  PROC DrawPart12()
    MoveL Offs(pOrigin,319.92,43.79,0.00),v40,z0,tPen\WObj:=wPaper;
    MoveL Offs(pOrigin,319.60,42.83,0.00),v40,z0,tPen\WObj:=wPaper;
    MoveL Offs(pOrigin,310.98,31.34,0.00),v40,z0,tPen\WObj:=wPaper;
    MoveL Offs(pOrigin,310.98,30.86,0.00),v40,z0,tPen\WObj:=wPaper;
    MoveL Offs(pOrigin,311.77,30.38,0.00),v40,z0,tPen\WObj:=wPaper;
    MoveL Offs(pOrigin,318.48,30.38,0.00),v40,z0,tPen\WObj:=wPaper;
    MoveL Offs(pOrigin,319.44,30.06,0.00),v40,z0,tPen\WObj:=wPaper;
    MoveL Offs(pOrigin,319.92,29.42,0.00),v40,z0,tPen\WObj:=wPaper;
    MoveL Offs(pOrigin,319.92,27.51,0.00),v40,z0,tPen\WObj:=wPaper;
    MoveL Offs(pOrigin,319.44,26.87,0.00),v40,z0,tPen\WObj:=wPaper;
    MoveL Offs(pOrigin,318.48,26.55,0.00),v40,z0,tPen\WObj:=wPaper;
    MoveL Offs(pOrigin,306.51,26.55,0.00),v40,z0,tPen\WObj:=wPaper;
    MoveL Offs(pOrigin,304.75,27.19,0.00),v40,z0,tPen\WObj:=wPaper;
    MoveL Offs(pOrigin,304.75,29.90,0.00),v40,z0,tPen\WObj:=wPaper;
    MoveL Offs(pOrigin,313.85,41.87,0.00),v40,z0,tPen\WObj:=wPaper;
    MoveL Offs(pOrigin,313.69,42.67,0.00),v40,z0,tPen\WObj:=wPaper;
    MoveL Offs(pOrigin,310.34,42.83,0.00),v40,z0,tPen\WObj:=wPaper;
    MoveL Offs(pOrigin,308.90,43.31,0.00),v40,z0,tPen\WObj:=wPaper;
    MoveL Offs(pOrigin,305.71,43.47,0.00),v40,z0,tPen\WObj:=wPaper;
    MoveL Offs(pOrigin,305.07,44.75,0.00),v40,fine,tPen\WObj:=wPaper;
    MoveL Offs(pOrigin,305.07,44.75,6.00),v60,z5,tPen\WObj:=wPaper;
    MoveL Offs(pOrigin,312.25,39.96,6.00),vTravel,z5,tPen\WObj:=wPaper;
    MoveL Offs(pOrigin,312.25,39.96,0.00),v60,z0,tPen\WObj:=wPaper;
    MoveL Offs(pOrigin,312.73,39.96,0.00),v40,z0,tPen\WObj:=wPaper;
    MoveL Offs(pOrigin,313.69,40.92,0.00),v40,z0,tPen\WObj:=wPaper;
    MoveL Offs(pOrigin,312.25,39.48,0.00),v40,z0,tPen\WObj:=wPaper;
    MoveL Offs(pOrigin,312.25,39.96,0.00),v40,z0,tPen\WObj:=wPaper;
    MoveL Offs(pOrigin,312.73,39.96,0.00),v40,z0,tPen\WObj:=wPaper;
    MoveL Offs(pOrigin,313.69,40.92,0.00),v40,z0,tPen\WObj:=wPaper;
    MoveL Offs(pOrigin,312.25,39.48,0.00),v40,z0,tPen\WObj:=wPaper;
    MoveL Offs(pOrigin,312.25,39.96,0.00),v40,fine,tPen\WObj:=wPaper;
    MoveL Offs(pOrigin,312.25,39.96,6.00),v60,z5,tPen\WObj:=wPaper;
    MoveL Offs(pOrigin,311.77,38.52,6.00),vTravel,z5,tPen\WObj:=wPaper;
    MoveL Offs(pOrigin,311.77,38.52,0.00),v60,z0,tPen\WObj:=wPaper;
    MoveL Offs(pOrigin,311.30,38.04,0.00),v40,z0,tPen\WObj:=wPaper;
    MoveL Offs(pOrigin,311.30,38.52,0.00),v40,z0,tPen\WObj:=wPaper;
    MoveL Offs(pOrigin,311.77,38.52,0.00),v40,z0,tPen\WObj:=wPaper;
    MoveL Offs(pOrigin,311.30,38.04,0.00),v40,z0,tPen\WObj:=wPaper;
    MoveL Offs(pOrigin,311.30,38.52,0.00),v40,z0,tPen\WObj:=wPaper;
    MoveL Offs(pOrigin,311.77,38.52,0.00),v40,fine,tPen\WObj:=wPaper;
    MoveL Offs(pOrigin,311.77,38.52,6.00),v60,z5,tPen\WObj:=wPaper;
    MoveL Offs(pOrigin,310.82,37.08,6.00),vTravel,z5,tPen\WObj:=wPaper;
    MoveL Offs(pOrigin,310.82,37.08,0.00),v60,z0,tPen\WObj:=wPaper;
    MoveL Offs(pOrigin,310.34,36.61,0.00),v40,z0,tPen\WObj:=wPaper;
    MoveL Offs(pOrigin,310.34,37.08,0.00),v40,z0,tPen\WObj:=wPaper;
    MoveL Offs(pOrigin,310.82,37.08,0.00),v40,z0,tPen\WObj:=wPaper;
    MoveL Offs(pOrigin,310.34,36.61,0.00),v40,z0,tPen\WObj:=wPaper;
    MoveL Offs(pOrigin,310.34,37.08,0.00),v40,z0,tPen\WObj:=wPaper;
    MoveL Offs(pOrigin,310.82,37.08,0.00),v40,fine,tPen\WObj:=wPaper;
    MoveL Offs(pOrigin,310.82,37.08,6.00),v60,z5,tPen\WObj:=wPaper;
    MoveL Offs(pOrigin,309.86,35.65,6.00),vTravel,z5,tPen\WObj:=wPaper;
    MoveL Offs(pOrigin,309.86,35.65,0.00),v60,z0,tPen\WObj:=wPaper;
    MoveL Offs(pOrigin,309.38,35.17,0.00),v40,z0,tPen\WObj:=wPaper;
    MoveL Offs(pOrigin,309.38,35.65,0.00),v40,z0,tPen\WObj:=wPaper;
    MoveL Offs(pOrigin,309.86,35.65,0.00),v40,z0,tPen\WObj:=wPaper;
    MoveL Offs(pOrigin,309.38,35.17,0.00),v40,z0,tPen\WObj:=wPaper;
    MoveL Offs(pOrigin,309.38,35.65,0.00),v40,z0,tPen\WObj:=wPaper;
    MoveL Offs(pOrigin,309.86,35.65,0.00),v40,fine,tPen\WObj:=wPaper;
    MoveL Offs(pOrigin,309.86,35.65,6.00),v60,z5,tPen\WObj:=wPaper;
    MoveL Offs(pOrigin,312.25,33.73,6.00),vTravel,z5,tPen\WObj:=wPaper;
    MoveL Offs(pOrigin,312.25,33.73,0.00),v60,z0,tPen\WObj:=wPaper;
    MoveL Offs(pOrigin,313.21,34.69,0.00),v40,z0,tPen\WObj:=wPaper;
    MoveL Offs(pOrigin,312.25,33.73,0.00),v40,z0,tPen\WObj:=wPaper;
    MoveL Offs(pOrigin,311.77,33.25,0.00),v40,z0,tPen\WObj:=wPaper;
    MoveL Offs(pOrigin,311.30,32.30,0.00),v40,z0,tPen\WObj:=wPaper;
    MoveL Offs(pOrigin,311.77,32.77,0.00),v40,z0,tPen\WObj:=wPaper;
    MoveL Offs(pOrigin,311.77,33.25,0.00),v40,z0,tPen\WObj:=wPaper;
    MoveL Offs(pOrigin,311.30,32.30,0.00),v40,z0,tPen\WObj:=wPaper;
    MoveL Offs(pOrigin,311.77,32.77,0.00),v40,z0,tPen\WObj:=wPaper;
    MoveL Offs(pOrigin,311.77,33.25,0.00),v40,fine,tPen\WObj:=wPaper;
    MoveL Offs(pOrigin,311.77,33.25,6.00),v60,z5,tPen\WObj:=wPaper;
    MoveL Offs(pOrigin,314.17,36.13,6.00),vTravel,z5,tPen\WObj:=wPaper;
    MoveL Offs(pOrigin,314.17,36.13,0.00),v60,z0,tPen\WObj:=wPaper;
    MoveL Offs(pOrigin,314.65,36.61,0.00),v40,z0,tPen\WObj:=wPaper;
    MoveL Offs(pOrigin,314.65,37.08,0.00),v40,z0,tPen\WObj:=wPaper;
    MoveL Offs(pOrigin,316.08,38.52,0.00),v40,z0,tPen\WObj:=wPaper;
    MoveL Offs(pOrigin,314.17,36.13,0.00),v40,z0,tPen\WObj:=wPaper;
    MoveL Offs(pOrigin,314.65,36.61,0.00),v40,z0,tPen\WObj:=wPaper;
    MoveL Offs(pOrigin,314.65,37.08,0.00),v40,z0,tPen\WObj:=wPaper;
    MoveL Offs(pOrigin,316.08,38.52,0.00),v40,z0,tPen\WObj:=wPaper;
    MoveL Offs(pOrigin,314.17,36.13,0.00),v40,fine,tPen\WObj:=wPaper;
    MoveL Offs(pOrigin,314.17,36.13,6.00),v60,z5,tPen\WObj:=wPaper;
    MoveL Offs(pOrigin,317.52,40.92,6.00),vTravel,z5,tPen\WObj:=wPaper;
    MoveL Offs(pOrigin,317.52,40.92,0.00),v60,z0,tPen\WObj:=wPaper;
    MoveL Offs(pOrigin,318.96,42.35,0.00),v40,z0,tPen\WObj:=wPaper;
    MoveL Offs(pOrigin,317.52,40.92,0.00),v40,fine,tPen\WObj:=wPaper;
    MoveL Offs(pOrigin,317.52,40.92,6.00),v60,z5,tPen\WObj:=wPaper;
    MoveL Offs(pOrigin,307.94,33.25,6.00),vTravel,z5,tPen\WObj:=wPaper;
    MoveL Offs(pOrigin,307.94,33.25,0.00),v60,z0,tPen\WObj:=wPaper;
    MoveL Offs(pOrigin,306.99,32.30,0.00),v40,z0,tPen\WObj:=wPaper;
    MoveL Offs(pOrigin,306.99,32.77,0.00),v40,z0,tPen\WObj:=wPaper;
    MoveL Offs(pOrigin,307.46,32.77,0.00),v40,z0,tPen\WObj:=wPaper;
    MoveL Offs(pOrigin,307.94,33.25,0.00),v40,z0,tPen\WObj:=wPaper;
    MoveL Offs(pOrigin,306.99,32.30,0.00),v40,z0,tPen\WObj:=wPaper;
    MoveL Offs(pOrigin,306.99,32.77,0.00),v40,z0,tPen\WObj:=wPaper;
    MoveL Offs(pOrigin,307.46,32.77,0.00),v40,z0,tPen\WObj:=wPaper;
    MoveL Offs(pOrigin,307.94,33.25,0.00),v40,fine,tPen\WObj:=wPaper;
    MoveL Offs(pOrigin,307.94,33.25,6.00),v60,z5,tPen\WObj:=wPaper;
    MoveL Offs(pOrigin,306.51,31.34,6.00),vTravel,z5,tPen\WObj:=wPaper;
    MoveL Offs(pOrigin,306.51,31.34,0.00),v60,z0,tPen\WObj:=wPaper;
    MoveL Offs(pOrigin,306.03,30.86,0.00),v40,z0,tPen\WObj:=wPaper;
    MoveL Offs(pOrigin,306.03,31.34,0.00),v40,z0,tPen\WObj:=wPaper;
    MoveL Offs(pOrigin,306.51,31.34,0.00),v40,z0,tPen\WObj:=wPaper;
    MoveL Offs(pOrigin,306.03,30.86,0.00),v40,z0,tPen\WObj:=wPaper;
    MoveL Offs(pOrigin,306.03,31.34,0.00),v40,z0,tPen\WObj:=wPaper;
    MoveL Offs(pOrigin,306.51,31.34,0.00),v40,fine,tPen\WObj:=wPaper;
    MoveL Offs(pOrigin,306.51,31.34,6.00),v60,z5,tPen\WObj:=wPaper;
    MoveL Offs(pOrigin,329.01,28.46,6.00),vTravel,z5,tPen\WObj:=wPaper;
    MoveL Offs(pOrigin,329.01,28.46,0.00),v60,z0,tPen\WObj:=wPaper;
    MoveL Offs(pOrigin,333.48,39.00,0.00),v40,z0,tPen\WObj:=wPaper;
    MoveL Offs(pOrigin,334.12,41.39,0.00),v40,z0,tPen\WObj:=wPaper;
    MoveL Offs(pOrigin,335.88,45.23,0.00),v40,z0,tPen\WObj:=wPaper;
    MoveL Offs(pOrigin,337.15,46.34,0.00),v40,z0,tPen\WObj:=wPaper;
    MoveL Offs(pOrigin,339.55,46.66,0.00),v40,z0,tPen\WObj:=wPaper;
    MoveL Offs(pOrigin,340.83,45.70,0.00),v40,z0,tPen\WObj:=wPaper;
    MoveL Offs(pOrigin,346.41,31.82,0.00),v40,z0,tPen\WObj:=wPaper;
    MoveL Offs(pOrigin,347.69,27.99,0.00),v40,z0,tPen\WObj:=wPaper;
    MoveL Offs(pOrigin,347.21,26.87,0.00),v40,z0,tPen\WObj:=wPaper;
    MoveL Offs(pOrigin,345.77,26.55,0.00),v40,z0,tPen\WObj:=wPaper;
    MoveL Offs(pOrigin,344.34,27.19,0.00),v40,z0,tPen\WObj:=wPaper;
  ENDPROC

  PROC DrawPart13()
    MoveL Offs(pOrigin,343.06,29.90,0.00),v40,z0,tPen\WObj:=wPaper;
    MoveL Offs(pOrigin,342.42,30.38,0.00),v40,z0,tPen\WObj:=wPaper;
    MoveL Offs(pOrigin,340.03,30.38,0.00),v40,z0,tPen\WObj:=wPaper;
    MoveL Offs(pOrigin,338.59,30.86,0.00),v40,z0,tPen\WObj:=wPaper;
    MoveL Offs(pOrigin,335.72,30.86,0.00),v40,z0,tPen\WObj:=wPaper;
    MoveL Offs(pOrigin,333.80,29.90,0.00),v40,z0,tPen\WObj:=wPaper;
    MoveL Offs(pOrigin,332.69,27.51,0.00),v40,z0,tPen\WObj:=wPaper;
    MoveL Offs(pOrigin,331.89,26.87,0.00),v40,z0,tPen\WObj:=wPaper;
    MoveL Offs(pOrigin,330.45,26.55,0.00),v40,z0,tPen\WObj:=wPaper;
    MoveL Offs(pOrigin,329.17,27.19,0.00),v40,z0,tPen\WObj:=wPaper;
    MoveL Offs(pOrigin,329.01,28.46,0.00),v40,fine,tPen\WObj:=wPaper;
    MoveL Offs(pOrigin,329.01,28.46,6.00),v60,z5,tPen\WObj:=wPaper;
    MoveL Offs(pOrigin,331.41,33.73,6.00),vTravel,z5,tPen\WObj:=wPaper;
    MoveL Offs(pOrigin,331.41,33.73,0.00),v60,z0,tPen\WObj:=wPaper;
    MoveL Offs(pOrigin,331.41,34.21,0.00),v40,z0,tPen\WObj:=wPaper;
    MoveL Offs(pOrigin,331.89,34.69,0.00),v40,z0,tPen\WObj:=wPaper;
    MoveL Offs(pOrigin,331.41,33.73,0.00),v40,z0,tPen\WObj:=wPaper;
    MoveL Offs(pOrigin,331.41,34.21,0.00),v40,z0,tPen\WObj:=wPaper;
    MoveL Offs(pOrigin,331.89,34.69,0.00),v40,z0,tPen\WObj:=wPaper;
    MoveL Offs(pOrigin,331.41,33.73,0.00),v40,fine,tPen\WObj:=wPaper;
    MoveL Offs(pOrigin,331.41,33.73,6.00),v60,z5,tPen\WObj:=wPaper;
    MoveL Offs(pOrigin,335.72,34.21,6.00),vTravel,z5,tPen\WObj:=wPaper;
    MoveL Offs(pOrigin,335.72,34.21,0.00),v60,z0,tPen\WObj:=wPaper;
    MoveL Offs(pOrigin,335.72,35.17,0.00),v40,z0,tPen\WObj:=wPaper;
    MoveL Offs(pOrigin,337.79,40.44,0.00),v40,z0,tPen\WObj:=wPaper;
    MoveL Offs(pOrigin,338.59,40.76,0.00),v40,z0,tPen\WObj:=wPaper;
    MoveL Offs(pOrigin,339.55,39.48,0.00),v40,z0,tPen\WObj:=wPaper;
    MoveL Offs(pOrigin,340.51,36.13,0.00),v40,z0,tPen\WObj:=wPaper;
    MoveL Offs(pOrigin,340.51,34.69,0.00),v40,z0,tPen\WObj:=wPaper;
    MoveL Offs(pOrigin,340.03,34.05,0.00),v40,z0,tPen\WObj:=wPaper;
    MoveL Offs(pOrigin,339.07,33.73,0.00),v40,z0,tPen\WObj:=wPaper;
    MoveL Offs(pOrigin,336.20,33.73,0.00),v40,z0,tPen\WObj:=wPaper;
    MoveL Offs(pOrigin,335.72,34.21,0.00),v40,fine,tPen\WObj:=wPaper;
    MoveL Offs(pOrigin,335.72,34.21,6.00),v60,z5,tPen\WObj:=wPaper;
    MoveL Offs(pOrigin,314.65,83.06,6.00),vTravel,z5,tPen\WObj:=wPaper;
    MoveL Offs(pOrigin,314.65,83.06,0.00),v60,z0,tPen\WObj:=wPaper;
    MoveL Offs(pOrigin,314.65,83.54,0.00),v40,z0,tPen\WObj:=wPaper;
    MoveL Offs(pOrigin,315.13,83.54,0.00),v40,z0,tPen\WObj:=wPaper;
    MoveL Offs(pOrigin,314.65,83.06,0.00),v40,z0,tPen\WObj:=wPaper;
    MoveL Offs(pOrigin,314.65,83.54,0.00),v40,z0,tPen\WObj:=wPaper;
    MoveL Offs(pOrigin,315.13,83.54,0.00),v40,z0,tPen\WObj:=wPaper;
    MoveL Offs(pOrigin,314.65,83.06,0.00),v40,fine,tPen\WObj:=wPaper;
    MoveL Offs(pOrigin,314.65,83.06,6.00),v60,z5,tPen\WObj:=wPaper;
    MoveL Offs(pOrigin,319.92,86.89,6.00),vTravel,z5,tPen\WObj:=wPaper;
    MoveL Offs(pOrigin,319.92,86.89,0.00),v60,z0,tPen\WObj:=wPaper;
    MoveL Offs(pOrigin,319.92,87.37,0.00),v40,z0,tPen\WObj:=wPaper;
    MoveL Offs(pOrigin,320.39,87.37,0.00),v40,z0,tPen\WObj:=wPaper;
    MoveL Offs(pOrigin,319.92,86.89,0.00),v40,z0,tPen\WObj:=wPaper;
    MoveL Offs(pOrigin,319.92,87.37,0.00),v40,z0,tPen\WObj:=wPaper;
    MoveL Offs(pOrigin,320.39,87.37,0.00),v40,z0,tPen\WObj:=wPaper;
    MoveL Offs(pOrigin,319.92,86.89,0.00),v40,fine,tPen\WObj:=wPaper;
    MoveL Offs(pOrigin,319.92,86.89,6.00),v60,z5,tPen\WObj:=wPaper;
    MoveL Offs(pOrigin,322.79,88.80,6.00),vTravel,z5,tPen\WObj:=wPaper;
    MoveL Offs(pOrigin,322.79,88.80,0.00),v60,z0,tPen\WObj:=wPaper;
    MoveL Offs(pOrigin,322.79,89.28,0.00),v40,z0,tPen\WObj:=wPaper;
    MoveL Offs(pOrigin,323.27,89.28,0.00),v40,z0,tPen\WObj:=wPaper;
    MoveL Offs(pOrigin,324.23,90.24,0.00),v40,z0,tPen\WObj:=wPaper;
    MoveL Offs(pOrigin,322.79,88.80,0.00),v40,z0,tPen\WObj:=wPaper;
    MoveL Offs(pOrigin,322.79,89.28,0.00),v40,z0,tPen\WObj:=wPaper;
    MoveL Offs(pOrigin,323.27,89.28,0.00),v40,z0,tPen\WObj:=wPaper;
    MoveL Offs(pOrigin,324.23,90.24,0.00),v40,z0,tPen\WObj:=wPaper;
    MoveL Offs(pOrigin,322.79,88.80,0.00),v40,fine,tPen\WObj:=wPaper;
    MoveL Offs(pOrigin,322.79,88.80,6.00),v60,z5,tPen\WObj:=wPaper;
    MoveL Offs(pOrigin,325.66,91.20,6.00),vTravel,z5,tPen\WObj:=wPaper;
    MoveL Offs(pOrigin,325.66,91.20,0.00),v60,z0,tPen\WObj:=wPaper;
    MoveL Offs(pOrigin,325.66,91.68,0.00),v40,z0,tPen\WObj:=wPaper;
    MoveL Offs(pOrigin,326.14,91.68,0.00),v40,z0,tPen\WObj:=wPaper;
    MoveL Offs(pOrigin,326.62,92.15,0.00),v40,z0,tPen\WObj:=wPaper;
    MoveL Offs(pOrigin,325.66,91.20,0.00),v40,z0,tPen\WObj:=wPaper;
    MoveL Offs(pOrigin,325.66,91.68,0.00),v40,z0,tPen\WObj:=wPaper;
    MoveL Offs(pOrigin,326.14,91.68,0.00),v40,z0,tPen\WObj:=wPaper;
    MoveL Offs(pOrigin,326.62,92.15,0.00),v40,z0,tPen\WObj:=wPaper;
    MoveL Offs(pOrigin,325.66,91.20,0.00),v40,fine,tPen\WObj:=wPaper;
    MoveL Offs(pOrigin,325.66,91.20,6.00),v60,z5,tPen\WObj:=wPaper;
    MoveL Offs(pOrigin,329.01,94.07,6.00),vTravel,z5,tPen\WObj:=wPaper;
    MoveL Offs(pOrigin,329.01,94.07,0.00),v60,z0,tPen\WObj:=wPaper;
    MoveL Offs(pOrigin,329.01,94.55,0.00),v40,z0,tPen\WObj:=wPaper;
    MoveL Offs(pOrigin,329.49,94.55,0.00),v40,z0,tPen\WObj:=wPaper;
    MoveL Offs(pOrigin,329.97,95.03,0.00),v40,z0,tPen\WObj:=wPaper;
    MoveL Offs(pOrigin,329.01,94.07,0.00),v40,z0,tPen\WObj:=wPaper;
    MoveL Offs(pOrigin,329.01,94.55,0.00),v40,z0,tPen\WObj:=wPaper;
    MoveL Offs(pOrigin,329.49,94.55,0.00),v40,z0,tPen\WObj:=wPaper;
    MoveL Offs(pOrigin,329.97,95.03,0.00),v40,z0,tPen\WObj:=wPaper;
    MoveL Offs(pOrigin,329.01,94.07,0.00),v40,fine,tPen\WObj:=wPaper;
    MoveL Offs(pOrigin,329.01,94.07,6.00),v60,z5,tPen\WObj:=wPaper;
    MoveL Offs(pOrigin,331.09,95.83,6.00),vTravel,z5,tPen\WObj:=wPaper;
    MoveL Offs(pOrigin,331.09,95.83,0.00),v60,z0,tPen\WObj:=wPaper;
    MoveL Offs(pOrigin,335.24,99.82,0.00),v40,z0,tPen\WObj:=wPaper;
    MoveL Offs(pOrigin,331.09,95.83,0.00),v40,fine,tPen\WObj:=wPaper;
    MoveL Offs(pOrigin,331.09,95.83,6.00),v60,z5,tPen\WObj:=wPaper;
    MoveL Offs(pOrigin,336.68,101.25,6.00),vTravel,z5,tPen\WObj:=wPaper;
    MoveL Offs(pOrigin,336.68,101.25,0.00),v60,z0,tPen\WObj:=wPaper;
    MoveL Offs(pOrigin,336.68,101.73,0.00),v40,z0,tPen\WObj:=wPaper;
    MoveL Offs(pOrigin,337.15,101.73,0.00),v40,z0,tPen\WObj:=wPaper;
    MoveL Offs(pOrigin,340.03,104.61,0.00),v40,z0,tPen\WObj:=wPaper;
    MoveL Offs(pOrigin,336.68,101.25,0.00),v40,z0,tPen\WObj:=wPaper;
    MoveL Offs(pOrigin,336.68,101.73,0.00),v40,z0,tPen\WObj:=wPaper;
    MoveL Offs(pOrigin,337.15,101.73,0.00),v40,z0,tPen\WObj:=wPaper;
    MoveL Offs(pOrigin,340.03,104.61,0.00),v40,z0,tPen\WObj:=wPaper;
    MoveL Offs(pOrigin,336.68,101.25,0.00),v40,fine,tPen\WObj:=wPaper;
    MoveL Offs(pOrigin,336.68,101.25,6.00),v60,z5,tPen\WObj:=wPaper;
    MoveL Offs(pOrigin,340.51,105.08,6.00),vTravel,z5,tPen\WObj:=wPaper;
    MoveL Offs(pOrigin,340.51,105.08,0.00),v60,z0,tPen\WObj:=wPaper;
    MoveL Offs(pOrigin,340.51,105.56,0.00),v40,z0,tPen\WObj:=wPaper;
    MoveL Offs(pOrigin,340.99,105.56,0.00),v40,z0,tPen\WObj:=wPaper;
    MoveL Offs(pOrigin,341.94,106.52,0.00),v40,z0,tPen\WObj:=wPaper;
    MoveL Offs(pOrigin,340.51,105.08,0.00),v40,z0,tPen\WObj:=wPaper;
    MoveL Offs(pOrigin,340.51,105.56,0.00),v40,z0,tPen\WObj:=wPaper;
    MoveL Offs(pOrigin,340.99,105.56,0.00),v40,z0,tPen\WObj:=wPaper;
    MoveL Offs(pOrigin,341.94,106.52,0.00),v40,z0,tPen\WObj:=wPaper;
    MoveL Offs(pOrigin,340.51,105.08,0.00),v40,fine,tPen\WObj:=wPaper;
    MoveL Offs(pOrigin,340.51,105.08,6.00),v60,z5,tPen\WObj:=wPaper;
    MoveL Offs(pOrigin,342.90,107.96,6.00),vTravel,z5,tPen\WObj:=wPaper;
    MoveL Offs(pOrigin,342.90,107.96,0.00),v60,z0,tPen\WObj:=wPaper;
    MoveL Offs(pOrigin,342.90,108.44,0.00),v40,z0,tPen\WObj:=wPaper;
    MoveL Offs(pOrigin,343.38,108.44,0.00),v40,z0,tPen\WObj:=wPaper;
    MoveL Offs(pOrigin,343.86,108.92,0.00),v40,z0,tPen\WObj:=wPaper;
    MoveL Offs(pOrigin,342.90,107.96,0.00),v40,z0,tPen\WObj:=wPaper;
    MoveL Offs(pOrigin,342.90,108.44,0.00),v40,z0,tPen\WObj:=wPaper;
    MoveL Offs(pOrigin,343.38,108.44,0.00),v40,z0,tPen\WObj:=wPaper;
  ENDPROC

  PROC DrawPart14()
    MoveL Offs(pOrigin,343.86,108.92,0.00),v40,z0,tPen\WObj:=wPaper;
    MoveL Offs(pOrigin,342.90,107.96,0.00),v40,fine,tPen\WObj:=wPaper;
    MoveL Offs(pOrigin,342.90,107.96,6.00),v60,z5,tPen\WObj:=wPaper;
    MoveL Offs(pOrigin,345.77,111.31,6.00),vTravel,z5,tPen\WObj:=wPaper;
    MoveL Offs(pOrigin,345.77,111.31,0.00),v60,z0,tPen\WObj:=wPaper;
    MoveL Offs(pOrigin,345.77,111.79,0.00),v40,z0,tPen\WObj:=wPaper;
    MoveL Offs(pOrigin,347.21,113.23,0.00),v40,z0,tPen\WObj:=wPaper;
    MoveL Offs(pOrigin,345.77,111.31,0.00),v40,z0,tPen\WObj:=wPaper;
    MoveL Offs(pOrigin,345.77,111.79,0.00),v40,z0,tPen\WObj:=wPaper;
    MoveL Offs(pOrigin,347.21,113.23,0.00),v40,z0,tPen\WObj:=wPaper;
    MoveL Offs(pOrigin,345.77,111.31,0.00),v40,fine,tPen\WObj:=wPaper;
    MoveL Offs(pOrigin,345.77,111.31,6.00),v60,z5,tPen\WObj:=wPaper;
    MoveL Offs(pOrigin,347.69,113.70,6.00),vTravel,z5,tPen\WObj:=wPaper;
    MoveL Offs(pOrigin,347.69,113.70,0.00),v60,z0,tPen\WObj:=wPaper;
    MoveL Offs(pOrigin,347.69,114.18,0.00),v40,z0,tPen\WObj:=wPaper;
    MoveL Offs(pOrigin,348.65,115.14,0.00),v40,z0,tPen\WObj:=wPaper;
    MoveL Offs(pOrigin,347.69,113.70,0.00),v40,z0,tPen\WObj:=wPaper;
    MoveL Offs(pOrigin,347.69,114.18,0.00),v40,z0,tPen\WObj:=wPaper;
    MoveL Offs(pOrigin,348.65,115.14,0.00),v40,z0,tPen\WObj:=wPaper;
    MoveL Offs(pOrigin,347.69,113.70,0.00),v40,fine,tPen\WObj:=wPaper;
    MoveL Offs(pOrigin,347.69,113.70,6.00),v60,z5,tPen\WObj:=wPaper;
    MoveL Offs(pOrigin,349.13,116.10,6.00),vTravel,z5,tPen\WObj:=wPaper;
    MoveL Offs(pOrigin,349.13,116.10,0.00),v60,z0,tPen\WObj:=wPaper;
    MoveL Offs(pOrigin,349.13,116.58,0.00),v40,z0,tPen\WObj:=wPaper;
    MoveL Offs(pOrigin,349.61,116.58,0.00),v40,z0,tPen\WObj:=wPaper;
    MoveL Offs(pOrigin,350.08,117.06,0.00),v40,z0,tPen\WObj:=wPaper;
    MoveL Offs(pOrigin,349.13,116.10,0.00),v40,z0,tPen\WObj:=wPaper;
    MoveL Offs(pOrigin,349.13,116.58,0.00),v40,z0,tPen\WObj:=wPaper;
    MoveL Offs(pOrigin,349.61,116.58,0.00),v40,z0,tPen\WObj:=wPaper;
    MoveL Offs(pOrigin,350.08,117.06,0.00),v40,z0,tPen\WObj:=wPaper;
    MoveL Offs(pOrigin,349.13,116.10,0.00),v40,fine,tPen\WObj:=wPaper;
    MoveL Offs(pOrigin,349.13,116.10,6.00),v60,z5,tPen\WObj:=wPaper;
    MoveL Offs(pOrigin,350.56,118.01,6.00),vTravel,z5,tPen\WObj:=wPaper;
    MoveL Offs(pOrigin,350.56,118.01,0.00),v60,z0,tPen\WObj:=wPaper;
    MoveL Offs(pOrigin,350.56,118.49,0.00),v40,z0,tPen\WObj:=wPaper;
    MoveL Offs(pOrigin,351.04,118.49,0.00),v40,z0,tPen\WObj:=wPaper;
    MoveL Offs(pOrigin,350.56,118.01,0.00),v40,z0,tPen\WObj:=wPaper;
    MoveL Offs(pOrigin,350.56,118.49,0.00),v40,z0,tPen\WObj:=wPaper;
    MoveL Offs(pOrigin,351.04,118.49,0.00),v40,z0,tPen\WObj:=wPaper;
    MoveL Offs(pOrigin,350.56,118.01,0.00),v40,fine,tPen\WObj:=wPaper;
    MoveL Offs(pOrigin,350.56,118.01,6.00),v60,z5,tPen\WObj:=wPaper;
    MoveL Offs(pOrigin,351.52,119.45,6.00),vTravel,z5,tPen\WObj:=wPaper;
    MoveL Offs(pOrigin,351.52,119.45,0.00),v60,z0,tPen\WObj:=wPaper;
    MoveL Offs(pOrigin,351.52,119.93,0.00),v40,z0,tPen\WObj:=wPaper;
    MoveL Offs(pOrigin,352.00,119.93,0.00),v40,z0,tPen\WObj:=wPaper;
    MoveL Offs(pOrigin,351.52,119.45,0.00),v40,z0,tPen\WObj:=wPaper;
    MoveL Offs(pOrigin,351.52,119.93,0.00),v40,z0,tPen\WObj:=wPaper;
    MoveL Offs(pOrigin,352.00,119.93,0.00),v40,z0,tPen\WObj:=wPaper;
    MoveL Offs(pOrigin,351.52,119.45,0.00),v40,fine,tPen\WObj:=wPaper;
    MoveL Offs(pOrigin,351.52,119.45,6.00),v60,z5,tPen\WObj:=wPaper;
    MoveL Offs(pOrigin,352.48,120.89,6.00),vTravel,z5,tPen\WObj:=wPaper;
    MoveL Offs(pOrigin,352.48,120.89,0.00),v60,z0,tPen\WObj:=wPaper;
    MoveL Offs(pOrigin,352.48,121.37,0.00),v40,z0,tPen\WObj:=wPaper;
    MoveL Offs(pOrigin,352.96,121.37,0.00),v40,z0,tPen\WObj:=wPaper;
    MoveL Offs(pOrigin,352.48,120.89,0.00),v40,z0,tPen\WObj:=wPaper;
    MoveL Offs(pOrigin,352.48,121.37,0.00),v40,z0,tPen\WObj:=wPaper;
    MoveL Offs(pOrigin,352.96,121.37,0.00),v40,z0,tPen\WObj:=wPaper;
    MoveL Offs(pOrigin,352.48,120.89,0.00),v40,fine,tPen\WObj:=wPaper;
    MoveL Offs(pOrigin,352.48,120.89,6.00),v60,z5,tPen\WObj:=wPaper;
    MoveL Offs(pOrigin,355.83,126.15,6.00),vTravel,z5,tPen\WObj:=wPaper;
    MoveL Offs(pOrigin,355.83,126.15,0.00),v60,z0,tPen\WObj:=wPaper;
    MoveL Offs(pOrigin,355.83,126.63,0.00),v40,z0,tPen\WObj:=wPaper;
    MoveL Offs(pOrigin,356.31,127.11,0.00),v40,z0,tPen\WObj:=wPaper;
    MoveL Offs(pOrigin,355.83,126.15,0.00),v40,z0,tPen\WObj:=wPaper;
    MoveL Offs(pOrigin,355.83,126.63,0.00),v40,z0,tPen\WObj:=wPaper;
    MoveL Offs(pOrigin,356.31,127.11,0.00),v40,z0,tPen\WObj:=wPaper;
    MoveL Offs(pOrigin,355.83,126.15,0.00),v40,fine,tPen\WObj:=wPaper;
    MoveL Offs(pOrigin,355.83,126.15,6.00),v60,z5,tPen\WObj:=wPaper;
    MoveL Offs(pOrigin,357.27,129.03,6.00),vTravel,z5,tPen\WObj:=wPaper;
    MoveL Offs(pOrigin,357.27,129.03,0.00),v60,z0,tPen\WObj:=wPaper;
    MoveL Offs(pOrigin,357.27,129.51,0.00),v40,z0,tPen\WObj:=wPaper;
    MoveL Offs(pOrigin,357.75,129.51,0.00),v40,z0,tPen\WObj:=wPaper;
    MoveL Offs(pOrigin,357.27,129.03,0.00),v40,z0,tPen\WObj:=wPaper;
    MoveL Offs(pOrigin,357.27,129.51,0.00),v40,z0,tPen\WObj:=wPaper;
    MoveL Offs(pOrigin,357.75,129.51,0.00),v40,z0,tPen\WObj:=wPaper;
    MoveL Offs(pOrigin,357.27,129.03,0.00),v40,fine,tPen\WObj:=wPaper;
    MoveL Offs(pOrigin,357.27,129.03,6.00),v60,z5,tPen\WObj:=wPaper;
    MoveL Offs(pOrigin,358.23,130.46,6.00),vTravel,z5,tPen\WObj:=wPaper;
    MoveL Offs(pOrigin,358.23,130.46,0.00),v60,z0,tPen\WObj:=wPaper;
    MoveL Offs(pOrigin,358.23,130.94,0.00),v40,z0,tPen\WObj:=wPaper;
    MoveL Offs(pOrigin,358.70,131.42,0.00),v40,z0,tPen\WObj:=wPaper;
    MoveL Offs(pOrigin,358.23,130.46,0.00),v40,z0,tPen\WObj:=wPaper;
    MoveL Offs(pOrigin,358.23,130.94,0.00),v40,z0,tPen\WObj:=wPaper;
    MoveL Offs(pOrigin,358.70,131.42,0.00),v40,z0,tPen\WObj:=wPaper;
    MoveL Offs(pOrigin,358.23,130.46,0.00),v40,fine,tPen\WObj:=wPaper;
    MoveL Offs(pOrigin,358.23,130.46,6.00),v60,z5,tPen\WObj:=wPaper;
    MoveL Offs(pOrigin,359.18,132.38,6.00),vTravel,z5,tPen\WObj:=wPaper;
    MoveL Offs(pOrigin,359.18,132.38,0.00),v60,z0,tPen\WObj:=wPaper;
    MoveL Offs(pOrigin,359.18,132.86,0.00),v40,z0,tPen\WObj:=wPaper;
    MoveL Offs(pOrigin,359.66,132.86,0.00),v40,z0,tPen\WObj:=wPaper;
    MoveL Offs(pOrigin,359.18,132.38,0.00),v40,z0,tPen\WObj:=wPaper;
    MoveL Offs(pOrigin,359.18,132.86,0.00),v40,z0,tPen\WObj:=wPaper;
    MoveL Offs(pOrigin,359.66,132.86,0.00),v40,z0,tPen\WObj:=wPaper;
    MoveL Offs(pOrigin,359.18,132.38,0.00),v40,fine,tPen\WObj:=wPaper;
    MoveL Offs(pOrigin,359.18,132.38,6.00),v60,z5,tPen\WObj:=wPaper;
    MoveL Offs(pOrigin,361.10,136.21,6.00),vTravel,z5,tPen\WObj:=wPaper;
    MoveL Offs(pOrigin,361.10,136.21,0.00),v60,z0,tPen\WObj:=wPaper;
    MoveL Offs(pOrigin,361.10,136.69,0.00),v40,z0,tPen\WObj:=wPaper;
    MoveL Offs(pOrigin,361.58,137.17,0.00),v40,z0,tPen\WObj:=wPaper;
    MoveL Offs(pOrigin,361.10,136.21,0.00),v40,z0,tPen\WObj:=wPaper;
    MoveL Offs(pOrigin,361.10,136.69,0.00),v40,z0,tPen\WObj:=wPaper;
    MoveL Offs(pOrigin,361.58,137.17,0.00),v40,z0,tPen\WObj:=wPaper;
    MoveL Offs(pOrigin,361.10,136.21,0.00),v40,fine,tPen\WObj:=wPaper;
    MoveL Offs(pOrigin,361.10,136.21,6.00),v60,z5,tPen\WObj:=wPaper;
    MoveL Offs(pOrigin,353.44,138.61,6.00),vTravel,z5,tPen\WObj:=wPaper;
    MoveL Offs(pOrigin,353.44,138.61,0.00),v60,z0,tPen\WObj:=wPaper;
    MoveL Offs(pOrigin,353.44,139.08,0.00),v40,z0,tPen\WObj:=wPaper;
    MoveL Offs(pOrigin,352.96,138.13,0.00),v40,z0,tPen\WObj:=wPaper;
    MoveL Offs(pOrigin,353.44,138.61,0.00),v40,z0,tPen\WObj:=wPaper;
    MoveL Offs(pOrigin,353.44,139.08,0.00),v40,z0,tPen\WObj:=wPaper;
    MoveL Offs(pOrigin,352.96,138.13,0.00),v40,z0,tPen\WObj:=wPaper;
    MoveL Offs(pOrigin,353.44,138.61,0.00),v40,fine,tPen\WObj:=wPaper;
    MoveL Offs(pOrigin,353.44,138.61,6.00),v60,z5,tPen\WObj:=wPaper;
    MoveL Offs(pOrigin,352.00,136.21,6.00),vTravel,z5,tPen\WObj:=wPaper;
    MoveL Offs(pOrigin,352.00,136.21,0.00),v60,z0,tPen\WObj:=wPaper;
    MoveL Offs(pOrigin,351.52,135.25,0.00),v40,z0,tPen\WObj:=wPaper;
    MoveL Offs(pOrigin,352.00,135.73,0.00),v40,z0,tPen\WObj:=wPaper;
    MoveL Offs(pOrigin,352.00,136.21,0.00),v40,z0,tPen\WObj:=wPaper;
    MoveL Offs(pOrigin,351.52,135.25,0.00),v40,z0,tPen\WObj:=wPaper;
    MoveL Offs(pOrigin,352.00,135.73,0.00),v40,z0,tPen\WObj:=wPaper;
  ENDPROC

  PROC DrawPart15()
    MoveL Offs(pOrigin,352.00,136.21,0.00),v40,fine,tPen\WObj:=wPaper;
    MoveL Offs(pOrigin,352.00,136.21,6.00),v60,z5,tPen\WObj:=wPaper;
    MoveL Offs(pOrigin,349.13,130.94,6.00),vTravel,z5,tPen\WObj:=wPaper;
    MoveL Offs(pOrigin,349.13,130.94,0.00),v60,z0,tPen\WObj:=wPaper;
    MoveL Offs(pOrigin,348.65,129.99,0.00),v40,z0,tPen\WObj:=wPaper;
    MoveL Offs(pOrigin,349.13,130.46,0.00),v40,z0,tPen\WObj:=wPaper;
    MoveL Offs(pOrigin,349.13,130.94,0.00),v40,z0,tPen\WObj:=wPaper;
    MoveL Offs(pOrigin,348.65,129.99,0.00),v40,z0,tPen\WObj:=wPaper;
    MoveL Offs(pOrigin,349.13,130.46,0.00),v40,z0,tPen\WObj:=wPaper;
    MoveL Offs(pOrigin,349.13,130.94,0.00),v40,fine,tPen\WObj:=wPaper;
    MoveL Offs(pOrigin,349.13,130.94,6.00),v60,z5,tPen\WObj:=wPaper;
    MoveL Offs(pOrigin,346.25,126.15,6.00),vTravel,z5,tPen\WObj:=wPaper;
    MoveL Offs(pOrigin,346.25,126.15,0.00),v60,z0,tPen\WObj:=wPaper;
    MoveL Offs(pOrigin,347.21,127.59,0.00),v40,z0,tPen\WObj:=wPaper;
    MoveL Offs(pOrigin,346.25,126.15,0.00),v40,fine,tPen\WObj:=wPaper;
    MoveL Offs(pOrigin,346.25,126.15,6.00),v60,z5,tPen\WObj:=wPaper;
    MoveL Offs(pOrigin,344.82,124.24,6.00),vTravel,z5,tPen\WObj:=wPaper;
    MoveL Offs(pOrigin,344.82,124.24,0.00),v60,z0,tPen\WObj:=wPaper;
    MoveL Offs(pOrigin,345.77,125.20,0.00),v40,z0,tPen\WObj:=wPaper;
    MoveL Offs(pOrigin,344.82,124.24,0.00),v40,fine,tPen\WObj:=wPaper;
    MoveL Offs(pOrigin,344.82,124.24,6.00),v60,z5,tPen\WObj:=wPaper;
    MoveL Offs(pOrigin,342.90,121.37,6.00),vTravel,z5,tPen\WObj:=wPaper;
    MoveL Offs(pOrigin,342.90,121.37,0.00),v60,z0,tPen\WObj:=wPaper;
    MoveL Offs(pOrigin,343.86,122.32,0.00),v40,z0,tPen\WObj:=wPaper;
    MoveL Offs(pOrigin,342.90,121.37,0.00),v40,fine,tPen\WObj:=wPaper;
    MoveL Offs(pOrigin,342.90,121.37,6.00),v60,z5,tPen\WObj:=wPaper;
    MoveL Offs(pOrigin,341.46,119.45,6.00),vTravel,z5,tPen\WObj:=wPaper;
    MoveL Offs(pOrigin,341.46,119.45,0.00),v60,z0,tPen\WObj:=wPaper;
    MoveL Offs(pOrigin,342.42,120.41,0.00),v40,z0,tPen\WObj:=wPaper;
    MoveL Offs(pOrigin,341.46,119.45,0.00),v40,fine,tPen\WObj:=wPaper;
    MoveL Offs(pOrigin,341.46,119.45,6.00),v60,z5,tPen\WObj:=wPaper;
    MoveL Offs(pOrigin,339.55,116.58,6.00),vTravel,z5,tPen\WObj:=wPaper;
    MoveL Offs(pOrigin,339.55,116.58,0.00),v60,z0,tPen\WObj:=wPaper;
    MoveL Offs(pOrigin,340.99,118.49,0.00),v40,z0,tPen\WObj:=wPaper;
    MoveL Offs(pOrigin,339.55,116.58,0.00),v40,fine,tPen\WObj:=wPaper;
    MoveL Offs(pOrigin,339.55,116.58,6.00),v60,z5,tPen\WObj:=wPaper;
    MoveL Offs(pOrigin,338.11,115.14,6.00),vTravel,z5,tPen\WObj:=wPaper;
    MoveL Offs(pOrigin,338.11,115.14,0.00),v60,z0,tPen\WObj:=wPaper;
    MoveL Offs(pOrigin,339.07,116.10,0.00),v40,z0,tPen\WObj:=wPaper;
    MoveL Offs(pOrigin,338.11,115.14,0.00),v40,fine,tPen\WObj:=wPaper;
    MoveL Offs(pOrigin,338.11,115.14,6.00),v60,z5,tPen\WObj:=wPaper;
    MoveL Offs(pOrigin,336.20,112.75,6.00),vTravel,z5,tPen\WObj:=wPaper;
    MoveL Offs(pOrigin,336.20,112.75,0.00),v60,z0,tPen\WObj:=wPaper;
    MoveL Offs(pOrigin,337.15,113.70,0.00),v40,z0,tPen\WObj:=wPaper;
    MoveL Offs(pOrigin,336.20,112.75,0.00),v40,fine,tPen\WObj:=wPaper;
    MoveL Offs(pOrigin,336.20,112.75,6.00),v60,z5,tPen\WObj:=wPaper;
    MoveL Offs(pOrigin,333.80,109.87,6.00),vTravel,z5,tPen\WObj:=wPaper;
    MoveL Offs(pOrigin,333.80,109.87,0.00),v60,z0,tPen\WObj:=wPaper;
    MoveL Offs(pOrigin,335.24,111.31,0.00),v40,z0,tPen\WObj:=wPaper;
    MoveL Offs(pOrigin,333.80,109.87,0.00),v40,fine,tPen\WObj:=wPaper;
    MoveL Offs(pOrigin,333.80,109.87,6.00),v60,z5,tPen\WObj:=wPaper;
    MoveL Offs(pOrigin,328.54,104.61,6.00),vTravel,z5,tPen\WObj:=wPaper;
    MoveL Offs(pOrigin,328.54,104.61,0.00),v60,z0,tPen\WObj:=wPaper;
    MoveL Offs(pOrigin,333.32,109.39,0.00),v40,z0,tPen\WObj:=wPaper;
    MoveL Offs(pOrigin,328.54,104.61,0.00),v40,fine,tPen\WObj:=wPaper;
    MoveL Offs(pOrigin,328.54,104.61,6.00),v60,z5,tPen\WObj:=wPaper;
    MoveL Offs(pOrigin,325.18,101.25,6.00),vTravel,z5,tPen\WObj:=wPaper;
    MoveL Offs(pOrigin,325.18,101.25,0.00),v60,z0,tPen\WObj:=wPaper;
    MoveL Offs(pOrigin,327.58,103.65,0.00),v40,z0,tPen\WObj:=wPaper;
    MoveL Offs(pOrigin,325.18,101.25,0.00),v40,fine,tPen\WObj:=wPaper;
    MoveL Offs(pOrigin,325.18,101.25,6.00),v60,z5,tPen\WObj:=wPaper;
    MoveL Offs(pOrigin,320.39,97.42,6.00),vTravel,z5,tPen\WObj:=wPaper;
    MoveL Offs(pOrigin,320.39,97.42,0.00),v60,z0,tPen\WObj:=wPaper;
    MoveL Offs(pOrigin,321.83,98.86,0.00),v40,z0,tPen\WObj:=wPaper;
    MoveL Offs(pOrigin,320.39,97.42,0.00),v40,fine,tPen\WObj:=wPaper;
    MoveL Offs(pOrigin,320.39,97.42,6.00),v60,z5,tPen\WObj:=wPaper;
    MoveL Offs(pOrigin,315.13,104.61,6.00),vTravel,z5,tPen\WObj:=wPaper;
    MoveL Offs(pOrigin,315.13,104.61,0.00),v60,z0,tPen\WObj:=wPaper;
    MoveL Offs(pOrigin,312.73,102.21,0.00),v40,z0,tPen\WObj:=wPaper;
    MoveL Offs(pOrigin,312.73,102.69,0.00),v40,z0,tPen\WObj:=wPaper;
    MoveL Offs(pOrigin,313.21,102.69,0.00),v40,z0,tPen\WObj:=wPaper;
    MoveL Offs(pOrigin,315.13,104.61,0.00),v40,z0,tPen\WObj:=wPaper;
    MoveL Offs(pOrigin,312.73,102.21,0.00),v40,z0,tPen\WObj:=wPaper;
    MoveL Offs(pOrigin,312.73,102.69,0.00),v40,z0,tPen\WObj:=wPaper;
    MoveL Offs(pOrigin,313.21,102.69,0.00),v40,z0,tPen\WObj:=wPaper;
    MoveL Offs(pOrigin,315.13,104.61,0.00),v40,fine,tPen\WObj:=wPaper;
    MoveL Offs(pOrigin,315.13,104.61,6.00),v60,z5,tPen\WObj:=wPaper;
    MoveL Offs(pOrigin,307.94,98.38,6.00),vTravel,z5,tPen\WObj:=wPaper;
    MoveL Offs(pOrigin,307.94,98.38,0.00),v60,z0,tPen\WObj:=wPaper;
    MoveL Offs(pOrigin,307.46,97.90,0.00),v40,z0,tPen\WObj:=wPaper;
    MoveL Offs(pOrigin,307.46,98.38,0.00),v40,z0,tPen\WObj:=wPaper;
    MoveL Offs(pOrigin,307.94,98.38,0.00),v40,z0,tPen\WObj:=wPaper;
    MoveL Offs(pOrigin,307.46,97.90,0.00),v40,z0,tPen\WObj:=wPaper;
    MoveL Offs(pOrigin,307.46,98.38,0.00),v40,z0,tPen\WObj:=wPaper;
    MoveL Offs(pOrigin,307.94,98.38,0.00),v40,fine,tPen\WObj:=wPaper;
    MoveL Offs(pOrigin,307.94,98.38,6.00),v60,z5,tPen\WObj:=wPaper;
    MoveL Offs(pOrigin,304.59,95.99,6.00),vTravel,z5,tPen\WObj:=wPaper;
    MoveL Offs(pOrigin,304.59,95.99,0.00),v60,z0,tPen\WObj:=wPaper;
    MoveL Offs(pOrigin,304.11,95.51,0.00),v40,z0,tPen\WObj:=wPaper;
    MoveL Offs(pOrigin,304.11,95.99,0.00),v40,z0,tPen\WObj:=wPaper;
    MoveL Offs(pOrigin,304.59,95.99,0.00),v40,z0,tPen\WObj:=wPaper;
    MoveL Offs(pOrigin,304.11,95.51,0.00),v40,z0,tPen\WObj:=wPaper;
    MoveL Offs(pOrigin,304.11,95.99,0.00),v40,z0,tPen\WObj:=wPaper;
    MoveL Offs(pOrigin,304.59,95.99,0.00),v40,fine,tPen\WObj:=wPaper;
    MoveL Offs(pOrigin,304.59,95.99,6.00),v60,z5,tPen\WObj:=wPaper;
    MoveL Offs(pOrigin,302.68,101.25,6.00),vTravel,z5,tPen\WObj:=wPaper;
    MoveL Offs(pOrigin,302.68,101.25,0.00),v60,z0,tPen\WObj:=wPaper;
    MoveL Offs(pOrigin,303.63,102.21,0.00),v40,z0,tPen\WObj:=wPaper;
    MoveL Offs(pOrigin,302.20,101.25,0.00),v40,z0,tPen\WObj:=wPaper;
    MoveL Offs(pOrigin,302.68,101.25,0.00),v40,z0,tPen\WObj:=wPaper;
    MoveL Offs(pOrigin,303.63,102.21,0.00),v40,z0,tPen\WObj:=wPaper;
    MoveL Offs(pOrigin,302.20,101.25,0.00),v40,z0,tPen\WObj:=wPaper;
    MoveL Offs(pOrigin,302.68,101.25,0.00),v40,fine,tPen\WObj:=wPaper;
    MoveL Offs(pOrigin,302.68,101.25,6.00),v60,z5,tPen\WObj:=wPaper;
    MoveL Offs(pOrigin,304.11,102.69,6.00),vTravel,z5,tPen\WObj:=wPaper;
    MoveL Offs(pOrigin,304.11,102.69,0.00),v60,z0,tPen\WObj:=wPaper;
    MoveL Offs(pOrigin,304.59,102.69,0.00),v40,z0,tPen\WObj:=wPaper;
    MoveL Offs(pOrigin,305.55,103.65,0.00),v40,z0,tPen\WObj:=wPaper;
    MoveL Offs(pOrigin,304.11,102.69,0.00),v40,z0,tPen\WObj:=wPaper;
    MoveL Offs(pOrigin,304.59,102.69,0.00),v40,z0,tPen\WObj:=wPaper;
    MoveL Offs(pOrigin,305.55,103.65,0.00),v40,z0,tPen\WObj:=wPaper;
    MoveL Offs(pOrigin,304.11,102.69,0.00),v40,fine,tPen\WObj:=wPaper;
    MoveL Offs(pOrigin,304.11,102.69,6.00),v60,z5,tPen\WObj:=wPaper;
    MoveL Offs(pOrigin,299.32,99.34,6.00),vTravel,z5,tPen\WObj:=wPaper;
    MoveL Offs(pOrigin,299.32,99.34,0.00),v60,z0,tPen\WObj:=wPaper;
    MoveL Offs(pOrigin,297.89,98.38,0.00),v40,z0,tPen\WObj:=wPaper;
    MoveL Offs(pOrigin,298.37,98.38,0.00),v40,z0,tPen\WObj:=wPaper;
    MoveL Offs(pOrigin,299.32,99.34,0.00),v40,z0,tPen\WObj:=wPaper;
    MoveL Offs(pOrigin,297.89,98.38,0.00),v40,z0,tPen\WObj:=wPaper;
    MoveL Offs(pOrigin,298.37,98.38,0.00),v40,z0,tPen\WObj:=wPaper;
  ENDPROC

  PROC DrawPart16()
    MoveL Offs(pOrigin,299.32,99.34,0.00),v40,fine,tPen\WObj:=wPaper;
    MoveL Offs(pOrigin,299.32,99.34,6.00),v60,z5,tPen\WObj:=wPaper;
    MoveL Offs(pOrigin,296.93,97.90,6.00),vTravel,z5,tPen\WObj:=wPaper;
    MoveL Offs(pOrigin,296.93,97.90,0.00),v60,z0,tPen\WObj:=wPaper;
    MoveL Offs(pOrigin,295.49,96.94,0.00),v40,z0,tPen\WObj:=wPaper;
    MoveL Offs(pOrigin,295.97,96.94,0.00),v40,z0,tPen\WObj:=wPaper;
    MoveL Offs(pOrigin,296.93,97.90,0.00),v40,z0,tPen\WObj:=wPaper;
    MoveL Offs(pOrigin,295.49,96.94,0.00),v40,z0,tPen\WObj:=wPaper;
    MoveL Offs(pOrigin,295.97,96.94,0.00),v40,z0,tPen\WObj:=wPaper;
    MoveL Offs(pOrigin,296.93,97.90,0.00),v40,fine,tPen\WObj:=wPaper;
    MoveL Offs(pOrigin,296.93,97.90,6.00),v60,z5,tPen\WObj:=wPaper;
    MoveL Offs(pOrigin,294.54,96.46,6.00),vTravel,z5,tPen\WObj:=wPaper;
    MoveL Offs(pOrigin,294.54,96.46,0.00),v60,z0,tPen\WObj:=wPaper;
    MoveL Offs(pOrigin,293.58,95.99,0.00),v40,z0,tPen\WObj:=wPaper;
    MoveL Offs(pOrigin,294.06,95.99,0.00),v40,z0,tPen\WObj:=wPaper;
    MoveL Offs(pOrigin,294.54,96.46,0.00),v40,z0,tPen\WObj:=wPaper;
    MoveL Offs(pOrigin,293.58,95.99,0.00),v40,z0,tPen\WObj:=wPaper;
    MoveL Offs(pOrigin,294.06,95.99,0.00),v40,z0,tPen\WObj:=wPaper;
    MoveL Offs(pOrigin,294.54,96.46,0.00),v40,fine,tPen\WObj:=wPaper;
    MoveL Offs(pOrigin,294.54,96.46,6.00),v60,z5,tPen\WObj:=wPaper;
    MoveL Offs(pOrigin,297.89,91.68,6.00),vTravel,z5,tPen\WObj:=wPaper;
    MoveL Offs(pOrigin,297.89,91.68,0.00),v60,z0,tPen\WObj:=wPaper;
    MoveL Offs(pOrigin,298.37,91.68,0.00),v40,z0,tPen\WObj:=wPaper;
    MoveL Offs(pOrigin,297.89,91.20,0.00),v40,z0,tPen\WObj:=wPaper;
    MoveL Offs(pOrigin,297.89,91.68,0.00),v40,z0,tPen\WObj:=wPaper;
    MoveL Offs(pOrigin,298.37,91.68,0.00),v40,z0,tPen\WObj:=wPaper;
    MoveL Offs(pOrigin,297.89,91.20,0.00),v40,z0,tPen\WObj:=wPaper;
    MoveL Offs(pOrigin,297.89,91.68,0.00),v40,fine,tPen\WObj:=wPaper;
    MoveL Offs(pOrigin,297.89,91.68,6.00),v60,z5,tPen\WObj:=wPaper;
    MoveL Offs(pOrigin,296.93,90.72,6.00),vTravel,z5,tPen\WObj:=wPaper;
    MoveL Offs(pOrigin,296.93,90.72,0.00),v60,z0,tPen\WObj:=wPaper;
    MoveL Offs(pOrigin,296.45,90.24,0.00),v40,z0,tPen\WObj:=wPaper;
    MoveL Offs(pOrigin,296.45,90.72,0.00),v40,z0,tPen\WObj:=wPaper;
    MoveL Offs(pOrigin,296.93,90.72,0.00),v40,z0,tPen\WObj:=wPaper;
    MoveL Offs(pOrigin,296.45,90.24,0.00),v40,z0,tPen\WObj:=wPaper;
    MoveL Offs(pOrigin,296.45,90.72,0.00),v40,z0,tPen\WObj:=wPaper;
    MoveL Offs(pOrigin,296.93,90.72,0.00),v40,fine,tPen\WObj:=wPaper;
    MoveL Offs(pOrigin,296.93,90.72,6.00),v60,z5,tPen\WObj:=wPaper;
    MoveL Offs(pOrigin,301.72,85.45,6.00),vTravel,z5,tPen\WObj:=wPaper;
    MoveL Offs(pOrigin,301.72,85.45,0.00),v60,z0,tPen\WObj:=wPaper;
    MoveL Offs(pOrigin,302.20,85.45,0.00),v40,z0,tPen\WObj:=wPaper;
    MoveL Offs(pOrigin,302.68,85.93,0.00),v40,z0,tPen\WObj:=wPaper;
    MoveL Offs(pOrigin,301.72,85.45,0.00),v40,z0,tPen\WObj:=wPaper;
    MoveL Offs(pOrigin,302.20,85.45,0.00),v40,z0,tPen\WObj:=wPaper;
    MoveL Offs(pOrigin,302.68,85.93,0.00),v40,z0,tPen\WObj:=wPaper;
    MoveL Offs(pOrigin,301.72,85.45,0.00),v40,fine,tPen\WObj:=wPaper;
    MoveL Offs(pOrigin,301.72,85.45,6.00),v60,z5,tPen\WObj:=wPaper;
    MoveL Offs(pOrigin,306.03,87.85,6.00),vTravel,z5,tPen\WObj:=wPaper;
    MoveL Offs(pOrigin,306.03,87.85,0.00),v60,z0,tPen\WObj:=wPaper;
    MoveL Offs(pOrigin,306.51,87.85,0.00),v40,z0,tPen\WObj:=wPaper;
    MoveL Offs(pOrigin,306.99,88.32,0.00),v40,z0,tPen\WObj:=wPaper;
    MoveL Offs(pOrigin,306.03,87.85,0.00),v40,z0,tPen\WObj:=wPaper;
    MoveL Offs(pOrigin,306.51,87.85,0.00),v40,z0,tPen\WObj:=wPaper;
    MoveL Offs(pOrigin,306.99,88.32,0.00),v40,z0,tPen\WObj:=wPaper;
    MoveL Offs(pOrigin,306.03,87.85,0.00),v40,fine,tPen\WObj:=wPaper;
    MoveL Offs(pOrigin,306.03,87.85,6.00),v60,z5,tPen\WObj:=wPaper;
    MoveL Offs(pOrigin,308.42,89.28,6.00),vTravel,z5,tPen\WObj:=wPaper;
    MoveL Offs(pOrigin,308.42,89.28,0.00),v60,z0,tPen\WObj:=wPaper;
    MoveL Offs(pOrigin,308.90,89.28,0.00),v40,z0,tPen\WObj:=wPaper;
    MoveL Offs(pOrigin,309.38,89.76,0.00),v40,z0,tPen\WObj:=wPaper;
    MoveL Offs(pOrigin,308.42,89.28,0.00),v40,z0,tPen\WObj:=wPaper;
    MoveL Offs(pOrigin,308.90,89.28,0.00),v40,z0,tPen\WObj:=wPaper;
    MoveL Offs(pOrigin,309.38,89.76,0.00),v40,z0,tPen\WObj:=wPaper;
    MoveL Offs(pOrigin,308.42,89.28,0.00),v40,fine,tPen\WObj:=wPaper;
    MoveL Offs(pOrigin,308.42,89.28,6.00),v60,z5,tPen\WObj:=wPaper;
    MoveL Offs(pOrigin,311.77,91.20,6.00),vTravel,z5,tPen\WObj:=wPaper;
    MoveL Offs(pOrigin,311.77,91.20,0.00),v60,z0,tPen\WObj:=wPaper;
    MoveL Offs(pOrigin,312.73,92.15,0.00),v40,z0,tPen\WObj:=wPaper;
    MoveL Offs(pOrigin,311.77,91.20,0.00),v40,fine,tPen\WObj:=wPaper;
    MoveL Offs(pOrigin,311.77,91.20,6.00),v60,z5,tPen\WObj:=wPaper;
    MoveL Offs(pOrigin,288.79,93.59,6.00),vTravel,z5,tPen\WObj:=wPaper;
    MoveL Offs(pOrigin,288.79,93.59,0.00),v60,z0,tPen\WObj:=wPaper;
    MoveL Offs(pOrigin,287.83,93.11,0.00),v40,z0,tPen\WObj:=wPaper;
    MoveL Offs(pOrigin,288.31,93.11,0.00),v40,z0,tPen\WObj:=wPaper;
    MoveL Offs(pOrigin,288.79,93.59,0.00),v40,z0,tPen\WObj:=wPaper;
    MoveL Offs(pOrigin,287.83,93.11,0.00),v40,z0,tPen\WObj:=wPaper;
    MoveL Offs(pOrigin,288.31,93.11,0.00),v40,z0,tPen\WObj:=wPaper;
    MoveL Offs(pOrigin,288.79,93.59,0.00),v40,fine,tPen\WObj:=wPaper;
    MoveL Offs(pOrigin,288.79,93.59,6.00),v60,z5,tPen\WObj:=wPaper;
    MoveL Offs(pOrigin,285.92,124.72,6.00),vTravel,z5,tPen\WObj:=wPaper;
    MoveL Offs(pOrigin,285.92,124.72,0.00),v60,z0,tPen\WObj:=wPaper;
    MoveL Offs(pOrigin,287.35,125.20,0.00),v40,z0,tPen\WObj:=wPaper;
    MoveL Offs(pOrigin,292.14,125.20,0.00),v40,z0,tPen\WObj:=wPaper;
    MoveL Offs(pOrigin,293.58,125.68,0.00),v40,z0,tPen\WObj:=wPaper;
    MoveL Offs(pOrigin,295.97,125.68,0.00),v40,z0,tPen\WObj:=wPaper;
    MoveL Offs(pOrigin,297.41,126.15,0.00),v40,z0,tPen\WObj:=wPaper;
    MoveL Offs(pOrigin,302.20,126.15,0.00),v40,z0,tPen\WObj:=wPaper;
    MoveL Offs(pOrigin,303.63,126.63,0.00),v40,z0,tPen\WObj:=wPaper;
    MoveL Offs(pOrigin,306.99,126.63,0.00),v40,z0,tPen\WObj:=wPaper;
    MoveL Offs(pOrigin,308.42,127.11,0.00),v40,z0,tPen\WObj:=wPaper;
    MoveL Offs(pOrigin,312.25,127.27,0.00),v40,z0,tPen\WObj:=wPaper;
    MoveL Offs(pOrigin,283.04,124.72,0.00),v40,z0,tPen\WObj:=wPaper;
    MoveL Offs(pOrigin,285.92,124.72,0.00),v40,fine,tPen\WObj:=wPaper;
    MoveL Offs(pOrigin,285.92,124.72,6.00),v60,z5,tPen\WObj:=wPaper;
    MoveL Offs(pOrigin,270.11,141.48,6.00),vTravel,z5,tPen\WObj:=wPaper;
    MoveL Offs(pOrigin,270.11,141.48,0.00),v60,z0,tPen\WObj:=wPaper;
    MoveL Offs(pOrigin,265.80,138.13,0.00),v40,z0,tPen\WObj:=wPaper;
    MoveL Offs(pOrigin,261.01,135.09,0.00),v40,z0,tPen\WObj:=wPaper;
    MoveL Offs(pOrigin,256.23,132.70,0.00),v40,z0,tPen\WObj:=wPaper;
    MoveL Offs(pOrigin,250.96,130.94,0.00),v40,z0,tPen\WObj:=wPaper;
    MoveL Offs(pOrigin,246.65,129.99,0.00),v40,z0,tPen\WObj:=wPaper;
    MoveL Offs(pOrigin,238.99,129.99,0.00),v40,z0,tPen\WObj:=wPaper;
    MoveL Offs(pOrigin,233.24,131.74,0.00),v40,z0,tPen\WObj:=wPaper;
    MoveL Offs(pOrigin,230.37,133.18,0.00),v40,z0,tPen\WObj:=wPaper;
    MoveL Offs(pOrigin,228.93,134.62,0.00),v40,z0,tPen\WObj:=wPaper;
    MoveL Offs(pOrigin,227.97,134.93,0.00),v40,z0,tPen\WObj:=wPaper;
    MoveL Offs(pOrigin,224.30,139.08,0.00),v40,z0,tPen\WObj:=wPaper;
    MoveL Offs(pOrigin,223.82,140.52,0.00),v40,z0,tPen\WObj:=wPaper;
    MoveL Offs(pOrigin,222.86,141.96,0.00),v40,z0,tPen\WObj:=wPaper;
    MoveL Offs(pOrigin,220.79,149.14,0.00),v40,z0,tPen\WObj:=wPaper;
    MoveL Offs(pOrigin,220.79,157.76,0.00),v40,z0,tPen\WObj:=wPaper;
    MoveL Offs(pOrigin,221.75,160.63,0.00),v40,z0,tPen\WObj:=wPaper;
    MoveL Offs(pOrigin,221.75,163.03,0.00),v40,z0,tPen\WObj:=wPaper;
    MoveL Offs(pOrigin,222.70,165.42,0.00),v40,z0,tPen\WObj:=wPaper;
    MoveL Offs(pOrigin,223.34,168.30,0.00),v40,z0,tPen\WObj:=wPaper;
    MoveL Offs(pOrigin,226.38,175.00,0.00),v40,z0,tPen\WObj:=wPaper;
    MoveL Offs(pOrigin,229.25,179.79,0.00),v40,z0,tPen\WObj:=wPaper;
    MoveL Offs(pOrigin,235.15,187.93,0.00),v40,z0,tPen\WObj:=wPaper;
    MoveL Offs(pOrigin,241.38,194.15,0.00),v40,z0,tPen\WObj:=wPaper;
    MoveL Offs(pOrigin,245.69,197.51,0.00),v40,z0,tPen\WObj:=wPaper;
  ENDPROC

  PROC DrawPart17()
    MoveL Offs(pOrigin,249.04,199.58,0.00),v40,z0,tPen\WObj:=wPaper;
    MoveL Offs(pOrigin,254.79,202.46,0.00),v40,z0,tPen\WObj:=wPaper;
    MoveL Offs(pOrigin,258.62,203.73,0.00),v40,z0,tPen\WObj:=wPaper;
    MoveL Offs(pOrigin,265.80,205.17,0.00),v40,z0,tPen\WObj:=wPaper;
    MoveL Offs(pOrigin,267.72,205.17,0.00),v40,z0,tPen\WObj:=wPaper;
    MoveL Offs(pOrigin,274.42,203.41,0.00),v40,z0,tPen\WObj:=wPaper;
    MoveL Offs(pOrigin,278.73,201.50,0.00),v40,z0,tPen\WObj:=wPaper;
    MoveL Offs(pOrigin,284.00,196.55,0.00),v40,z0,tPen\WObj:=wPaper;
    MoveL Offs(pOrigin,285.60,194.15,0.00),v40,z0,tPen\WObj:=wPaper;
    MoveL Offs(pOrigin,287.03,190.80,0.00),v40,z0,tPen\WObj:=wPaper;
    MoveL Offs(pOrigin,287.83,187.93,0.00),v40,z0,tPen\WObj:=wPaper;
    MoveL Offs(pOrigin,288.31,183.14,0.00),v40,z0,tPen\WObj:=wPaper;
    MoveL Offs(pOrigin,289.27,181.38,0.00),v40,z0,tPen\WObj:=wPaper;
    MoveL Offs(pOrigin,292.14,181.38,0.00),v40,z0,tPen\WObj:=wPaper;
    MoveL Offs(pOrigin,296.45,184.10,0.00),v40,z0,tPen\WObj:=wPaper;
    MoveL Offs(pOrigin,300.76,187.45,0.00),v40,z0,tPen\WObj:=wPaper;
    MoveL Offs(pOrigin,303.15,187.29,0.00),v40,z0,tPen\WObj:=wPaper;
    MoveL Offs(pOrigin,304.43,186.01,0.00),v40,z0,tPen\WObj:=wPaper;
    MoveL Offs(pOrigin,305.07,183.62,0.00),v40,z0,tPen\WObj:=wPaper;
    MoveL Offs(pOrigin,304.27,181.23,0.00),v40,z0,tPen\WObj:=wPaper;
    MoveL Offs(pOrigin,302.20,177.87,0.00),v40,z0,tPen\WObj:=wPaper;
    MoveL Offs(pOrigin,296.93,173.88,0.00),v40,z0,tPen\WObj:=wPaper;
    MoveL Offs(pOrigin,294.06,172.45,0.00),v40,z0,tPen\WObj:=wPaper;
    MoveL Offs(pOrigin,288.79,171.01,0.00),v40,z0,tPen\WObj:=wPaper;
    MoveL Offs(pOrigin,287.35,169.73,0.00),v40,z0,tPen\WObj:=wPaper;
    MoveL Offs(pOrigin,286.71,168.77,0.00),v40,z0,tPen\WObj:=wPaper;
    MoveL Offs(pOrigin,286.23,166.38,0.00),v40,z0,tPen\WObj:=wPaper;
    MoveL Offs(pOrigin,282.72,158.24,0.00),v40,z0,tPen\WObj:=wPaper;
    MoveL Offs(pOrigin,279.37,152.49,0.00),v40,z0,tPen\WObj:=wPaper;
    MoveL Offs(pOrigin,274.42,145.79,0.00),v40,z0,tPen\WObj:=wPaper;
    MoveL Offs(pOrigin,270.11,141.48,0.00),v40,z0,tPen\WObj:=wPaper;
    MoveL Offs(pOrigin,269.15,141.16,0.00),v40,z0,tPen\WObj:=wPaper;
    MoveL Offs(pOrigin,273.94,145.79,0.00),v40,z0,tPen\WObj:=wPaper;
    MoveL Offs(pOrigin,269.15,141.16,0.00),v40,fine,tPen\WObj:=wPaper;
    MoveL Offs(pOrigin,269.15,141.16,6.00),v60,z5,tPen\WObj:=wPaper;
    MoveL Offs(pOrigin,265.32,138.13,6.00),vTravel,z5,tPen\WObj:=wPaper;
    MoveL Offs(pOrigin,265.32,138.13,0.00),v60,z0,tPen\WObj:=wPaper;
    MoveL Offs(pOrigin,266.76,139.56,0.00),v40,z0,tPen\WObj:=wPaper;
    MoveL Offs(pOrigin,265.32,138.13,0.00),v40,fine,tPen\WObj:=wPaper;
    MoveL Offs(pOrigin,265.32,138.13,6.00),v60,z5,tPen\WObj:=wPaper;
    MoveL Offs(pOrigin,261.97,136.21,6.00),vTravel,z5,tPen\WObj:=wPaper;
    MoveL Offs(pOrigin,261.97,136.21,0.00),v60,z0,tPen\WObj:=wPaper;
    MoveL Offs(pOrigin,260.54,135.25,0.00),v40,z0,tPen\WObj:=wPaper;
    MoveL Offs(pOrigin,261.01,135.25,0.00),v40,z0,tPen\WObj:=wPaper;
    MoveL Offs(pOrigin,261.97,136.21,0.00),v40,z0,tPen\WObj:=wPaper;
    MoveL Offs(pOrigin,260.54,135.25,0.00),v40,z0,tPen\WObj:=wPaper;
    MoveL Offs(pOrigin,261.01,135.25,0.00),v40,z0,tPen\WObj:=wPaper;
    MoveL Offs(pOrigin,261.97,136.21,0.00),v40,fine,tPen\WObj:=wPaper;
    MoveL Offs(pOrigin,261.97,136.21,6.00),v60,z5,tPen\WObj:=wPaper;
    MoveL Offs(pOrigin,259.58,134.77,6.00),vTravel,z5,tPen\WObj:=wPaper;
    MoveL Offs(pOrigin,259.58,134.77,0.00),v60,z0,tPen\WObj:=wPaper;
    MoveL Offs(pOrigin,258.62,134.30,0.00),v40,z0,tPen\WObj:=wPaper;
    MoveL Offs(pOrigin,259.10,134.30,0.00),v40,z0,tPen\WObj:=wPaper;
    MoveL Offs(pOrigin,259.58,134.77,0.00),v40,z0,tPen\WObj:=wPaper;
    MoveL Offs(pOrigin,258.62,134.30,0.00),v40,z0,tPen\WObj:=wPaper;
    MoveL Offs(pOrigin,259.10,134.30,0.00),v40,z0,tPen\WObj:=wPaper;
    MoveL Offs(pOrigin,259.58,134.77,0.00),v40,fine,tPen\WObj:=wPaper;
    MoveL Offs(pOrigin,259.58,134.77,6.00),v60,z5,tPen\WObj:=wPaper;
    MoveL Offs(pOrigin,250.00,150.26,6.00),vTravel,z5,tPen\WObj:=wPaper;
    MoveL Offs(pOrigin,250.00,150.26,0.00),v60,z0,tPen\WObj:=wPaper;
    MoveL Offs(pOrigin,247.61,150.26,0.00),v40,z0,tPen\WObj:=wPaper;
    MoveL Offs(pOrigin,246.17,153.45,0.00),v40,z0,tPen\WObj:=wPaper;
    MoveL Offs(pOrigin,246.17,158.24,0.00),v40,z0,tPen\WObj:=wPaper;
    MoveL Offs(pOrigin,247.13,163.03,0.00),v40,z0,tPen\WObj:=wPaper;
    MoveL Offs(pOrigin,250.64,172.13,0.00),v40,z0,tPen\WObj:=wPaper;
    MoveL Offs(pOrigin,254.31,177.87,0.00),v40,z0,tPen\WObj:=wPaper;
    MoveL Offs(pOrigin,258.62,183.62,0.00),v40,z0,tPen\WObj:=wPaper;
    MoveL Offs(pOrigin,262.45,187.45,0.00),v40,z0,tPen\WObj:=wPaper;
    MoveL Offs(pOrigin,264.37,188.41,0.00),v40,z0,tPen\WObj:=wPaper;
    MoveL Offs(pOrigin,264.85,187.93,0.00),v40,z0,tPen\WObj:=wPaper;
    MoveL Offs(pOrigin,264.85,181.23,0.00),v40,z0,tPen\WObj:=wPaper;
    MoveL Offs(pOrigin,265.96,178.35,0.00),v40,z0,tPen\WObj:=wPaper;
    MoveL Offs(pOrigin,267.40,176.44,0.00),v40,z0,tPen\WObj:=wPaper;
    MoveL Offs(pOrigin,267.72,175.48,0.00),v40,z0,tPen\WObj:=wPaper;
    MoveL Offs(pOrigin,267.72,174.04,0.00),v40,z0,tPen\WObj:=wPaper;
    MoveL Offs(pOrigin,265.64,168.77,0.00),v40,z0,tPen\WObj:=wPaper;
    MoveL Offs(pOrigin,258.62,157.76,0.00),v40,z0,tPen\WObj:=wPaper;
    MoveL Offs(pOrigin,255.75,154.41,0.00),v40,z0,tPen\WObj:=wPaper;
    MoveL Offs(pOrigin,252.87,152.01,0.00),v40,z0,tPen\WObj:=wPaper;
    MoveL Offs(pOrigin,250.00,150.26,0.00),v40,fine,tPen\WObj:=wPaper;
    MoveL Offs(pOrigin,250.00,150.26,6.00),v60,z5,tPen\WObj:=wPaper;
    MoveL Offs(pOrigin,251.44,151.54,6.00),vTravel,z5,tPen\WObj:=wPaper;
    MoveL Offs(pOrigin,251.44,151.54,0.00),v60,z0,tPen\WObj:=wPaper;
    MoveL Offs(pOrigin,251.92,151.54,0.00),v40,z0,tPen\WObj:=wPaper;
    MoveL Offs(pOrigin,252.39,152.01,0.00),v40,z0,tPen\WObj:=wPaper;
    MoveL Offs(pOrigin,251.44,151.54,0.00),v40,z0,tPen\WObj:=wPaper;
    MoveL Offs(pOrigin,251.92,151.54,0.00),v40,z0,tPen\WObj:=wPaper;
    MoveL Offs(pOrigin,252.39,152.01,0.00),v40,z0,tPen\WObj:=wPaper;
    MoveL Offs(pOrigin,251.44,151.54,0.00),v40,fine,tPen\WObj:=wPaper;
    MoveL Offs(pOrigin,251.44,151.54,6.00),v60,z5,tPen\WObj:=wPaper;
    MoveL Offs(pOrigin,256.23,155.85,6.00),vTravel,z5,tPen\WObj:=wPaper;
    MoveL Offs(pOrigin,256.23,155.85,0.00),v60,z0,tPen\WObj:=wPaper;
    MoveL Offs(pOrigin,258.62,158.24,0.00),v40,z0,tPen\WObj:=wPaper;
    MoveL Offs(pOrigin,256.23,155.85,0.00),v40,fine,tPen\WObj:=wPaper;
    MoveL Offs(pOrigin,256.23,155.85,6.00),v60,z5,tPen\WObj:=wPaper;
    MoveL Offs(pOrigin,261.49,162.55,6.00),vTravel,z5,tPen\WObj:=wPaper;
    MoveL Offs(pOrigin,261.49,162.55,0.00),v60,z0,tPen\WObj:=wPaper;
    MoveL Offs(pOrigin,261.97,163.03,0.00),v40,z0,tPen\WObj:=wPaper;
    MoveL Offs(pOrigin,261.97,163.51,0.00),v40,z0,tPen\WObj:=wPaper;
    MoveL Offs(pOrigin,261.49,162.55,0.00),v40,z0,tPen\WObj:=wPaper;
    MoveL Offs(pOrigin,261.97,163.03,0.00),v40,z0,tPen\WObj:=wPaper;
    MoveL Offs(pOrigin,261.97,163.51,0.00),v40,z0,tPen\WObj:=wPaper;
    MoveL Offs(pOrigin,261.49,162.55,0.00),v40,fine,tPen\WObj:=wPaper;
    MoveL Offs(pOrigin,261.49,162.55,6.00),v60,z5,tPen\WObj:=wPaper;
    MoveL Offs(pOrigin,264.37,167.34,6.00),vTravel,z5,tPen\WObj:=wPaper;
    MoveL Offs(pOrigin,264.37,167.34,0.00),v60,z0,tPen\WObj:=wPaper;
    MoveL Offs(pOrigin,264.85,167.82,0.00),v40,z0,tPen\WObj:=wPaper;
    MoveL Offs(pOrigin,264.85,168.30,0.00),v40,z0,tPen\WObj:=wPaper;
    MoveL Offs(pOrigin,264.37,167.34,0.00),v40,z0,tPen\WObj:=wPaper;
    MoveL Offs(pOrigin,264.85,167.82,0.00),v40,z0,tPen\WObj:=wPaper;
    MoveL Offs(pOrigin,264.85,168.30,0.00),v40,z0,tPen\WObj:=wPaper;
    MoveL Offs(pOrigin,264.37,167.34,0.00),v40,fine,tPen\WObj:=wPaper;
    MoveL Offs(pOrigin,264.37,167.34,6.00),v60,z5,tPen\WObj:=wPaper;
    MoveL Offs(pOrigin,267.24,175.96,6.00),vTravel,z5,tPen\WObj:=wPaper;
    MoveL Offs(pOrigin,267.24,175.96,0.00),v60,z0,tPen\WObj:=wPaper;
    MoveL Offs(pOrigin,267.24,176.44,0.00),v40,z0,tPen\WObj:=wPaper;
    MoveL Offs(pOrigin,266.28,177.39,0.00),v40,z0,tPen\WObj:=wPaper;
    MoveL Offs(pOrigin,267.24,175.96,0.00),v40,z0,tPen\WObj:=wPaper;
    MoveL Offs(pOrigin,267.24,176.44,0.00),v40,z0,tPen\WObj:=wPaper;
    MoveL Offs(pOrigin,266.28,177.39,0.00),v40,z0,tPen\WObj:=wPaper;
  ENDPROC

  PROC DrawPart18()
    MoveL Offs(pOrigin,267.24,175.96,0.00),v40,fine,tPen\WObj:=wPaper;
    MoveL Offs(pOrigin,267.24,175.96,6.00),v60,z5,tPen\WObj:=wPaper;
    MoveL Offs(pOrigin,258.14,182.18,6.00),vTravel,z5,tPen\WObj:=wPaper;
    MoveL Offs(pOrigin,258.14,182.18,0.00),v60,z0,tPen\WObj:=wPaper;
    MoveL Offs(pOrigin,256.70,180.75,0.00),v40,z0,tPen\WObj:=wPaper;
    MoveL Offs(pOrigin,256.70,181.23,0.00),v40,z0,tPen\WObj:=wPaper;
    MoveL Offs(pOrigin,257.18,181.23,0.00),v40,z0,tPen\WObj:=wPaper;
    MoveL Offs(pOrigin,258.14,182.18,0.00),v40,z0,tPen\WObj:=wPaper;
    MoveL Offs(pOrigin,256.70,180.75,0.00),v40,z0,tPen\WObj:=wPaper;
    MoveL Offs(pOrigin,256.70,181.23,0.00),v40,z0,tPen\WObj:=wPaper;
    MoveL Offs(pOrigin,257.18,181.23,0.00),v40,z0,tPen\WObj:=wPaper;
    MoveL Offs(pOrigin,258.14,182.18,0.00),v40,fine,tPen\WObj:=wPaper;
    MoveL Offs(pOrigin,258.14,182.18,6.00),v60,z5,tPen\WObj:=wPaper;
    MoveL Offs(pOrigin,259.10,183.62,6.00),vTravel,z5,tPen\WObj:=wPaper;
    MoveL Offs(pOrigin,259.10,183.62,0.00),v60,z0,tPen\WObj:=wPaper;
    MoveL Offs(pOrigin,259.10,184.10,0.00),v40,z0,tPen\WObj:=wPaper;
    MoveL Offs(pOrigin,259.58,184.10,0.00),v40,z0,tPen\WObj:=wPaper;
    MoveL Offs(pOrigin,261.49,186.01,0.00),v40,z0,tPen\WObj:=wPaper;
    MoveL Offs(pOrigin,259.10,183.62,0.00),v40,z0,tPen\WObj:=wPaper;
    MoveL Offs(pOrigin,259.10,184.10,0.00),v40,z0,tPen\WObj:=wPaper;
    MoveL Offs(pOrigin,259.58,184.10,0.00),v40,z0,tPen\WObj:=wPaper;
    MoveL Offs(pOrigin,261.49,186.01,0.00),v40,z0,tPen\WObj:=wPaper;
    MoveL Offs(pOrigin,259.10,183.62,0.00),v40,fine,tPen\WObj:=wPaper;
    MoveL Offs(pOrigin,259.10,183.62,6.00),v60,z5,tPen\WObj:=wPaper;
    MoveL Offs(pOrigin,261.97,186.49,6.00),vTravel,z5,tPen\WObj:=wPaper;
    MoveL Offs(pOrigin,261.97,186.49,0.00),v60,z0,tPen\WObj:=wPaper;
    MoveL Offs(pOrigin,261.97,186.97,0.00),v40,z0,tPen\WObj:=wPaper;
    MoveL Offs(pOrigin,262.45,186.97,0.00),v40,z0,tPen\WObj:=wPaper;
    MoveL Offs(pOrigin,262.93,187.45,0.00),v40,z0,tPen\WObj:=wPaper;
    MoveL Offs(pOrigin,261.97,186.49,0.00),v40,z0,tPen\WObj:=wPaper;
    MoveL Offs(pOrigin,261.97,186.97,0.00),v40,z0,tPen\WObj:=wPaper;
    MoveL Offs(pOrigin,262.45,186.97,0.00),v40,z0,tPen\WObj:=wPaper;
    MoveL Offs(pOrigin,262.93,187.45,0.00),v40,z0,tPen\WObj:=wPaper;
    MoveL Offs(pOrigin,261.97,186.49,0.00),v40,fine,tPen\WObj:=wPaper;
    MoveL Offs(pOrigin,261.97,186.49,6.00),v60,z5,tPen\WObj:=wPaper;
    MoveL Offs(pOrigin,256.23,179.79,6.00),vTravel,z5,tPen\WObj:=wPaper;
    MoveL Offs(pOrigin,256.23,179.79,0.00),v60,z0,tPen\WObj:=wPaper;
    MoveL Offs(pOrigin,255.75,179.31,0.00),v40,z0,tPen\WObj:=wPaper;
    MoveL Offs(pOrigin,255.75,179.79,0.00),v40,z0,tPen\WObj:=wPaper;
    MoveL Offs(pOrigin,256.23,179.79,0.00),v40,z0,tPen\WObj:=wPaper;
    MoveL Offs(pOrigin,255.75,179.31,0.00),v40,z0,tPen\WObj:=wPaper;
    MoveL Offs(pOrigin,255.75,179.79,0.00),v40,z0,tPen\WObj:=wPaper;
    MoveL Offs(pOrigin,256.23,179.79,0.00),v40,fine,tPen\WObj:=wPaper;
    MoveL Offs(pOrigin,256.23,179.79,6.00),v60,z5,tPen\WObj:=wPaper;
    MoveL Offs(pOrigin,255.27,178.35,6.00),vTravel,z5,tPen\WObj:=wPaper;
    MoveL Offs(pOrigin,255.27,178.35,0.00),v60,z0,tPen\WObj:=wPaper;
    MoveL Offs(pOrigin,254.79,177.87,0.00),v40,z0,tPen\WObj:=wPaper;
    MoveL Offs(pOrigin,254.79,178.35,0.00),v40,z0,tPen\WObj:=wPaper;
    MoveL Offs(pOrigin,255.27,178.35,0.00),v40,z0,tPen\WObj:=wPaper;
    MoveL Offs(pOrigin,254.79,177.87,0.00),v40,z0,tPen\WObj:=wPaper;
    MoveL Offs(pOrigin,254.79,178.35,0.00),v40,z0,tPen\WObj:=wPaper;
    MoveL Offs(pOrigin,255.27,178.35,0.00),v40,fine,tPen\WObj:=wPaper;
    MoveL Offs(pOrigin,255.27,178.35,6.00),v60,z5,tPen\WObj:=wPaper;
    MoveL Offs(pOrigin,254.31,177.39,6.00),vTravel,z5,tPen\WObj:=wPaper;
    MoveL Offs(pOrigin,254.31,177.39,0.00),v60,z0,tPen\WObj:=wPaper;
    MoveL Offs(pOrigin,253.83,176.44,0.00),v40,z0,tPen\WObj:=wPaper;
    MoveL Offs(pOrigin,253.83,176.92,0.00),v40,z0,tPen\WObj:=wPaper;
    MoveL Offs(pOrigin,254.31,177.39,0.00),v40,z0,tPen\WObj:=wPaper;
    MoveL Offs(pOrigin,253.83,176.44,0.00),v40,z0,tPen\WObj:=wPaper;
    MoveL Offs(pOrigin,253.83,176.92,0.00),v40,z0,tPen\WObj:=wPaper;
    MoveL Offs(pOrigin,254.31,177.39,0.00),v40,fine,tPen\WObj:=wPaper;
    MoveL Offs(pOrigin,254.31,177.39,6.00),v60,z5,tPen\WObj:=wPaper;
    MoveL Offs(pOrigin,252.87,175.00,6.00),vTravel,z5,tPen\WObj:=wPaper;
    MoveL Offs(pOrigin,252.87,175.00,0.00),v60,z0,tPen\WObj:=wPaper;
    MoveL Offs(pOrigin,251.92,173.56,0.00),v40,z0,tPen\WObj:=wPaper;
    MoveL Offs(pOrigin,251.92,174.04,0.00),v40,z0,tPen\WObj:=wPaper;
    MoveL Offs(pOrigin,252.87,175.00,0.00),v40,z0,tPen\WObj:=wPaper;
    MoveL Offs(pOrigin,251.92,173.56,0.00),v40,z0,tPen\WObj:=wPaper;
    MoveL Offs(pOrigin,251.92,174.04,0.00),v40,z0,tPen\WObj:=wPaper;
    MoveL Offs(pOrigin,252.87,175.00,0.00),v40,fine,tPen\WObj:=wPaper;
    MoveL Offs(pOrigin,252.87,175.00,6.00),v60,z5,tPen\WObj:=wPaper;
    MoveL Offs(pOrigin,251.44,172.61,6.00),vTravel,z5,tPen\WObj:=wPaper;
    MoveL Offs(pOrigin,251.44,172.61,0.00),v60,z0,tPen\WObj:=wPaper;
    MoveL Offs(pOrigin,250.96,172.13,0.00),v40,z0,tPen\WObj:=wPaper;
    MoveL Offs(pOrigin,250.96,172.61,0.00),v40,z0,tPen\WObj:=wPaper;
    MoveL Offs(pOrigin,251.44,172.61,0.00),v40,z0,tPen\WObj:=wPaper;
    MoveL Offs(pOrigin,250.96,172.13,0.00),v40,z0,tPen\WObj:=wPaper;
    MoveL Offs(pOrigin,250.96,172.61,0.00),v40,z0,tPen\WObj:=wPaper;
    MoveL Offs(pOrigin,251.44,172.61,0.00),v40,fine,tPen\WObj:=wPaper;
    MoveL Offs(pOrigin,251.44,172.61,6.00),v60,z5,tPen\WObj:=wPaper;
    MoveL Offs(pOrigin,234.68,186.49,6.00),vTravel,z5,tPen\WObj:=wPaper;
    MoveL Offs(pOrigin,234.68,186.49,0.00),v60,z0,tPen\WObj:=wPaper;
    MoveL Offs(pOrigin,233.24,185.06,0.00),v40,z0,tPen\WObj:=wPaper;
    MoveL Offs(pOrigin,233.24,185.54,0.00),v40,z0,tPen\WObj:=wPaper;
    MoveL Offs(pOrigin,233.72,185.54,0.00),v40,z0,tPen\WObj:=wPaper;
    MoveL Offs(pOrigin,234.68,186.49,0.00),v40,z0,tPen\WObj:=wPaper;
    MoveL Offs(pOrigin,233.24,185.06,0.00),v40,z0,tPen\WObj:=wPaper;
    MoveL Offs(pOrigin,233.24,185.54,0.00),v40,z0,tPen\WObj:=wPaper;
    MoveL Offs(pOrigin,233.72,185.54,0.00),v40,z0,tPen\WObj:=wPaper;
    MoveL Offs(pOrigin,234.68,186.49,0.00),v40,z0,tPen\WObj:=wPaper;
    MoveL Offs(pOrigin,235.15,187.45,0.00),v40,z0,tPen\WObj:=wPaper;
    MoveL Offs(pOrigin,235.15,187.93,0.00),v40,z0,tPen\WObj:=wPaper;
    MoveL Offs(pOrigin,235.63,187.93,0.00),v40,z0,tPen\WObj:=wPaper;
    MoveL Offs(pOrigin,237.55,189.85,0.00),v40,z0,tPen\WObj:=wPaper;
    MoveL Offs(pOrigin,235.15,187.45,0.00),v40,z0,tPen\WObj:=wPaper;
    MoveL Offs(pOrigin,235.15,187.93,0.00),v40,z0,tPen\WObj:=wPaper;
    MoveL Offs(pOrigin,235.63,187.93,0.00),v40,z0,tPen\WObj:=wPaper;
    MoveL Offs(pOrigin,237.55,189.85,0.00),v40,z0,tPen\WObj:=wPaper;
    MoveL Offs(pOrigin,235.15,187.45,0.00),v40,fine,tPen\WObj:=wPaper;
    MoveL Offs(pOrigin,235.15,187.45,6.00),v60,z5,tPen\WObj:=wPaper;
    MoveL Offs(pOrigin,232.76,184.10,6.00),vTravel,z5,tPen\WObj:=wPaper;
    MoveL Offs(pOrigin,232.76,184.10,0.00),v60,z0,tPen\WObj:=wPaper;
    MoveL Offs(pOrigin,232.28,183.62,0.00),v40,z0,tPen\WObj:=wPaper;
    MoveL Offs(pOrigin,232.28,184.10,0.00),v40,z0,tPen\WObj:=wPaper;
    MoveL Offs(pOrigin,232.76,184.10,0.00),v40,z0,tPen\WObj:=wPaper;
    MoveL Offs(pOrigin,232.28,183.62,0.00),v40,z0,tPen\WObj:=wPaper;
    MoveL Offs(pOrigin,232.28,184.10,0.00),v40,z0,tPen\WObj:=wPaper;
    MoveL Offs(pOrigin,232.76,184.10,0.00),v40,fine,tPen\WObj:=wPaper;
    MoveL Offs(pOrigin,232.76,184.10,6.00),v60,z5,tPen\WObj:=wPaper;
    MoveL Offs(pOrigin,231.80,183.14,6.00),vTravel,z5,tPen\WObj:=wPaper;
    MoveL Offs(pOrigin,231.80,183.14,0.00),v60,z0,tPen\WObj:=wPaper;
    MoveL Offs(pOrigin,231.32,182.18,0.00),v40,z0,tPen\WObj:=wPaper;
    MoveL Offs(pOrigin,231.32,182.66,0.00),v40,z0,tPen\WObj:=wPaper;
    MoveL Offs(pOrigin,231.80,183.14,0.00),v40,z0,tPen\WObj:=wPaper;
    MoveL Offs(pOrigin,231.32,182.18,0.00),v40,z0,tPen\WObj:=wPaper;
    MoveL Offs(pOrigin,231.32,182.66,0.00),v40,z0,tPen\WObj:=wPaper;
    MoveL Offs(pOrigin,231.80,183.14,0.00),v40,fine,tPen\WObj:=wPaper;
    MoveL Offs(pOrigin,231.80,183.14,6.00),v60,z5,tPen\WObj:=wPaper;
    MoveL Offs(pOrigin,230.37,180.75,6.00),vTravel,z5,tPen\WObj:=wPaper;
    MoveL Offs(pOrigin,230.37,180.75,0.00),v60,z0,tPen\WObj:=wPaper;
  ENDPROC

  PROC DrawPart19()
    MoveL Offs(pOrigin,229.41,179.31,0.00),v40,z0,tPen\WObj:=wPaper;
    MoveL Offs(pOrigin,229.41,179.79,0.00),v40,z0,tPen\WObj:=wPaper;
    MoveL Offs(pOrigin,230.37,180.75,0.00),v40,z0,tPen\WObj:=wPaper;
    MoveL Offs(pOrigin,229.41,179.31,0.00),v40,z0,tPen\WObj:=wPaper;
    MoveL Offs(pOrigin,229.41,179.79,0.00),v40,z0,tPen\WObj:=wPaper;
    MoveL Offs(pOrigin,230.37,180.75,0.00),v40,fine,tPen\WObj:=wPaper;
    MoveL Offs(pOrigin,230.37,180.75,6.00),v60,z5,tPen\WObj:=wPaper;
    MoveL Offs(pOrigin,228.93,178.35,6.00),vTravel,z5,tPen\WObj:=wPaper;
    MoveL Offs(pOrigin,228.93,178.35,0.00),v60,z0,tPen\WObj:=wPaper;
    MoveL Offs(pOrigin,228.45,177.87,0.00),v40,z0,tPen\WObj:=wPaper;
    MoveL Offs(pOrigin,228.45,178.35,0.00),v40,z0,tPen\WObj:=wPaper;
    MoveL Offs(pOrigin,228.93,178.35,0.00),v40,z0,tPen\WObj:=wPaper;
    MoveL Offs(pOrigin,228.45,177.87,0.00),v40,z0,tPen\WObj:=wPaper;
    MoveL Offs(pOrigin,228.45,178.35,0.00),v40,z0,tPen\WObj:=wPaper;
    MoveL Offs(pOrigin,228.93,178.35,0.00),v40,fine,tPen\WObj:=wPaper;
    MoveL Offs(pOrigin,228.93,178.35,6.00),v60,z5,tPen\WObj:=wPaper;
    MoveL Offs(pOrigin,227.49,175.96,6.00),vTravel,z5,tPen\WObj:=wPaper;
    MoveL Offs(pOrigin,227.49,175.96,0.00),v60,z0,tPen\WObj:=wPaper;
    MoveL Offs(pOrigin,226.54,174.52,0.00),v40,z0,tPen\WObj:=wPaper;
    MoveL Offs(pOrigin,226.54,175.00,0.00),v40,z0,tPen\WObj:=wPaper;
    MoveL Offs(pOrigin,227.49,175.96,0.00),v40,z0,tPen\WObj:=wPaper;
    MoveL Offs(pOrigin,226.54,174.52,0.00),v40,z0,tPen\WObj:=wPaper;
    MoveL Offs(pOrigin,226.54,175.00,0.00),v40,z0,tPen\WObj:=wPaper;
    MoveL Offs(pOrigin,227.49,175.96,0.00),v40,fine,tPen\WObj:=wPaper;
    MoveL Offs(pOrigin,227.49,175.96,6.00),v60,z5,tPen\WObj:=wPaper;
    MoveL Offs(pOrigin,221.27,188.89,6.00),vTravel,z5,tPen\WObj:=wPaper;
    MoveL Offs(pOrigin,221.27,188.89,0.00),v60,z0,tPen\WObj:=wPaper;
    MoveL Offs(pOrigin,221.27,189.37,0.00),v40,z0,tPen\WObj:=wPaper;
    MoveL Offs(pOrigin,221.75,189.85,0.00),v40,z0,tPen\WObj:=wPaper;
    MoveL Offs(pOrigin,221.27,188.89,0.00),v40,z0,tPen\WObj:=wPaper;
    MoveL Offs(pOrigin,221.27,189.37,0.00),v40,z0,tPen\WObj:=wPaper;
    MoveL Offs(pOrigin,221.75,189.85,0.00),v40,z0,tPen\WObj:=wPaper;
    MoveL Offs(pOrigin,221.27,188.89,0.00),v40,fine,tPen\WObj:=wPaper;
    MoveL Offs(pOrigin,221.27,188.89,6.00),v60,z5,tPen\WObj:=wPaper;
    MoveL Offs(pOrigin,238.51,190.80,6.00),vTravel,z5,tPen\WObj:=wPaper;
    MoveL Offs(pOrigin,238.51,190.80,0.00),v60,z0,tPen\WObj:=wPaper;
    MoveL Offs(pOrigin,238.51,191.28,0.00),v40,z0,tPen\WObj:=wPaper;
    MoveL Offs(pOrigin,238.99,191.28,0.00),v40,z0,tPen\WObj:=wPaper;
    MoveL Offs(pOrigin,241.86,194.15,0.00),v40,z0,tPen\WObj:=wPaper;
    MoveL Offs(pOrigin,238.51,190.80,0.00),v40,z0,tPen\WObj:=wPaper;
    MoveL Offs(pOrigin,238.51,191.28,0.00),v40,z0,tPen\WObj:=wPaper;
    MoveL Offs(pOrigin,238.99,191.28,0.00),v40,z0,tPen\WObj:=wPaper;
    MoveL Offs(pOrigin,241.86,194.15,0.00),v40,z0,tPen\WObj:=wPaper;
    MoveL Offs(pOrigin,238.51,190.80,0.00),v40,fine,tPen\WObj:=wPaper;
    MoveL Offs(pOrigin,238.51,190.80,6.00),v60,z5,tPen\WObj:=wPaper;
    MoveL Offs(pOrigin,242.82,194.63,6.00),vTravel,z5,tPen\WObj:=wPaper;
    MoveL Offs(pOrigin,242.82,194.63,0.00),v60,z0,tPen\WObj:=wPaper;
    MoveL Offs(pOrigin,242.82,195.11,0.00),v40,z0,tPen\WObj:=wPaper;
    MoveL Offs(pOrigin,243.30,195.11,0.00),v40,z0,tPen\WObj:=wPaper;
    MoveL Offs(pOrigin,244.25,196.07,0.00),v40,z0,tPen\WObj:=wPaper;
    MoveL Offs(pOrigin,242.82,194.63,0.00),v40,z0,tPen\WObj:=wPaper;
    MoveL Offs(pOrigin,242.82,195.11,0.00),v40,z0,tPen\WObj:=wPaper;
    MoveL Offs(pOrigin,243.30,195.11,0.00),v40,z0,tPen\WObj:=wPaper;
    MoveL Offs(pOrigin,244.25,196.07,0.00),v40,z0,tPen\WObj:=wPaper;
    MoveL Offs(pOrigin,242.82,194.63,0.00),v40,fine,tPen\WObj:=wPaper;
    MoveL Offs(pOrigin,242.82,194.63,6.00),v60,z5,tPen\WObj:=wPaper;
    MoveL Offs(pOrigin,245.21,196.55,6.00),vTravel,z5,tPen\WObj:=wPaper;
    MoveL Offs(pOrigin,245.21,196.55,0.00),v60,z0,tPen\WObj:=wPaper;
    MoveL Offs(pOrigin,245.21,197.03,0.00),v40,z0,tPen\WObj:=wPaper;
    MoveL Offs(pOrigin,245.69,197.03,0.00),v40,z0,tPen\WObj:=wPaper;
    MoveL Offs(pOrigin,245.21,196.55,0.00),v40,z0,tPen\WObj:=wPaper;
    MoveL Offs(pOrigin,245.21,197.03,0.00),v40,z0,tPen\WObj:=wPaper;
    MoveL Offs(pOrigin,245.69,197.03,0.00),v40,z0,tPen\WObj:=wPaper;
    MoveL Offs(pOrigin,245.21,196.55,0.00),v40,fine,tPen\WObj:=wPaper;
    MoveL Offs(pOrigin,245.21,196.55,6.00),v60,z5,tPen\WObj:=wPaper;
    MoveL Offs(pOrigin,253.83,218.26,6.00),vTravel,z5,tPen\WObj:=wPaper;
    MoveL Offs(pOrigin,253.83,218.26,0.00),v60,z0,tPen\WObj:=wPaper;
    MoveL Offs(pOrigin,255.27,218.10,0.00),v40,z0,tPen\WObj:=wPaper;
    MoveL Offs(pOrigin,260.69,220.33,0.00),v40,z0,tPen\WObj:=wPaper;
    MoveL Offs(pOrigin,252.39,219.06,0.00),v40,z0,tPen\WObj:=wPaper;
    MoveL Offs(pOrigin,253.83,218.26,0.00),v40,fine,tPen\WObj:=wPaper;
    MoveL Offs(pOrigin,253.83,218.26,6.00),v60,z5,tPen\WObj:=wPaper;
    MoveL Offs(pOrigin,251.92,219.06,6.00),vTravel,z5,tPen\WObj:=wPaper;
    MoveL Offs(pOrigin,251.92,219.06,0.00),v60,z0,tPen\WObj:=wPaper;
    MoveL Offs(pOrigin,251.92,219.54,0.00),v40,z0,tPen\WObj:=wPaper;
    MoveL Offs(pOrigin,251.44,220.01,0.00),v40,z0,tPen\WObj:=wPaper;
    MoveL Offs(pOrigin,251.44,219.54,0.00),v40,z0,tPen\WObj:=wPaper;
    MoveL Offs(pOrigin,251.92,219.06,0.00),v40,z0,tPen\WObj:=wPaper;
    MoveL Offs(pOrigin,251.92,219.54,0.00),v40,z0,tPen\WObj:=wPaper;
    MoveL Offs(pOrigin,251.44,220.01,0.00),v40,z0,tPen\WObj:=wPaper;
    MoveL Offs(pOrigin,251.44,219.54,0.00),v40,z0,tPen\WObj:=wPaper;
    MoveL Offs(pOrigin,251.92,219.06,0.00),v40,fine,tPen\WObj:=wPaper;
    MoveL Offs(pOrigin,251.92,219.06,6.00),v60,z5,tPen\WObj:=wPaper;
    MoveL Offs(pOrigin,251.44,221.45,6.00),vTravel,z5,tPen\WObj:=wPaper;
    MoveL Offs(pOrigin,251.44,221.45,0.00),v60,z0,tPen\WObj:=wPaper;
    MoveL Offs(pOrigin,251.92,224.32,0.00),v40,z0,tPen\WObj:=wPaper;
    MoveL Offs(pOrigin,252.87,226.72,0.00),v40,z0,tPen\WObj:=wPaper;
    MoveL Offs(pOrigin,252.87,227.68,0.00),v40,z0,tPen\WObj:=wPaper;
    MoveL Offs(pOrigin,253.67,230.07,0.00),v40,z0,tPen\WObj:=wPaper;
    MoveL Offs(pOrigin,251.44,221.45,0.00),v40,fine,tPen\WObj:=wPaper;
    MoveL Offs(pOrigin,251.44,221.45,6.00),v60,z5,tPen\WObj:=wPaper;
    MoveL Offs(pOrigin,259.26,226.88,6.00),vTravel,z5,tPen\WObj:=wPaper;
    MoveL Offs(pOrigin,259.26,226.88,0.00),v60,z0,tPen\WObj:=wPaper;
    MoveL Offs(pOrigin,259.10,227.20,0.00),v40,z0,tPen\WObj:=wPaper;
    MoveL Offs(pOrigin,259.26,228.63,0.00),v40,z0,tPen\WObj:=wPaper;
    MoveL Offs(pOrigin,259.90,229.59,0.00),v40,z0,tPen\WObj:=wPaper;
    MoveL Offs(pOrigin,271.39,264.07,0.00),v40,z0,tPen\WObj:=wPaper;
    MoveL Offs(pOrigin,272.67,266.94,0.00),v40,z0,tPen\WObj:=wPaper;
    MoveL Offs(pOrigin,273.62,270.30,0.00),v40,z0,tPen\WObj:=wPaper;
    MoveL Offs(pOrigin,274.26,271.25,0.00),v40,z0,tPen\WObj:=wPaper;
    MoveL Offs(pOrigin,278.41,284.18,0.00),v40,z0,tPen\WObj:=wPaper;
    MoveL Offs(pOrigin,279.05,285.14,0.00),v40,z0,tPen\WObj:=wPaper;
    MoveL Offs(pOrigin,280.97,291.37,0.00),v40,z0,tPen\WObj:=wPaper;
    MoveL Offs(pOrigin,283.68,298.55,0.00),v40,z0,tPen\WObj:=wPaper;
    MoveL Offs(pOrigin,285.44,304.77,0.00),v40,z0,tPen\WObj:=wPaper;
    MoveL Offs(pOrigin,286.23,306.21,0.00),v40,z0,tPen\WObj:=wPaper;
    MoveL Offs(pOrigin,286.39,307.65,0.00),v40,z0,tPen\WObj:=wPaper;
    MoveL Offs(pOrigin,287.83,311.48,0.00),v40,z0,tPen\WObj:=wPaper;
    MoveL Offs(pOrigin,287.83,312.44,0.00),v40,z0,tPen\WObj:=wPaper;
    MoveL Offs(pOrigin,288.63,313.87,0.00),v40,z0,tPen\WObj:=wPaper;
    MoveL Offs(pOrigin,288.79,315.31,0.00),v40,z0,tPen\WObj:=wPaper;
    MoveL Offs(pOrigin,290.23,319.62,0.00),v40,z0,tPen\WObj:=wPaper;
    MoveL Offs(pOrigin,290.70,320.10,0.00),v40,z0,tPen\WObj:=wPaper;
    MoveL Offs(pOrigin,292.62,320.10,0.00),v40,z0,tPen\WObj:=wPaper;
    MoveL Offs(pOrigin,296.93,318.50,0.00),v40,z0,tPen\WObj:=wPaper;
    MoveL Offs(pOrigin,307.46,313.08,0.00),v40,z0,tPen\WObj:=wPaper;
    MoveL Offs(pOrigin,317.52,306.69,0.00),v40,z0,tPen\WObj:=wPaper;
    MoveL Offs(pOrigin,327.58,299.03,0.00),v40,z0,tPen\WObj:=wPaper;
    MoveL Offs(pOrigin,339.55,287.06,0.00),v40,z0,tPen\WObj:=wPaper;
    MoveL Offs(pOrigin,345.77,279.39,0.00),v40,z0,tPen\WObj:=wPaper;
  ENDPROC

  PROC DrawPart20()
    MoveL Offs(pOrigin,351.20,270.77,0.00),v40,z0,tPen\WObj:=wPaper;
    MoveL Offs(pOrigin,351.52,269.82,0.00),v40,z0,tPen\WObj:=wPaper;
    MoveL Offs(pOrigin,351.36,268.06,0.00),v40,z0,tPen\WObj:=wPaper;
    MoveL Offs(pOrigin,349.13,266.62,0.00),v40,z0,tPen\WObj:=wPaper;
    MoveL Offs(pOrigin,310.34,249.54,0.00),v40,z0,tPen\WObj:=wPaper;
    MoveL Offs(pOrigin,306.99,247.63,0.00),v40,z0,tPen\WObj:=wPaper;
    MoveL Offs(pOrigin,294.54,242.36,0.00),v40,z0,tPen\WObj:=wPaper;
    MoveL Offs(pOrigin,287.35,238.85,0.00),v40,z0,tPen\WObj:=wPaper;
    MoveL Offs(pOrigin,283.52,237.41,0.00),v40,z0,tPen\WObj:=wPaper;
    MoveL Offs(pOrigin,282.08,236.46,0.00),v40,z0,tPen\WObj:=wPaper;
    MoveL Offs(pOrigin,267.72,230.23,0.00),v40,z0,tPen\WObj:=wPaper;
    MoveL Offs(pOrigin,262.45,227.52,0.00),v40,z0,tPen\WObj:=wPaper;
    MoveL Offs(pOrigin,260.06,226.72,0.00),v40,z0,tPen\WObj:=wPaper;
    MoveL Offs(pOrigin,259.26,226.88,0.00),v40,fine,tPen\WObj:=wPaper;
    MoveL Offs(pOrigin,259.26,226.88,6.00),v60,z5,tPen\WObj:=wPaper;
    MoveL Offs(pOrigin,261.97,220.81,6.00),vTravel,z5,tPen\WObj:=wPaper;
    MoveL Offs(pOrigin,261.97,220.81,0.00),v60,z0,tPen\WObj:=wPaper;
    MoveL Offs(pOrigin,265.80,222.73,0.00),v40,z0,tPen\WObj:=wPaper;
    MoveL Offs(pOrigin,267.24,223.05,0.00),v40,z0,tPen\WObj:=wPaper;
    MoveL Offs(pOrigin,268.68,224.00,0.00),v40,z0,tPen\WObj:=wPaper;
    MoveL Offs(pOrigin,273.46,225.60,0.00),v40,z0,tPen\WObj:=wPaper;
    MoveL Offs(pOrigin,275.38,226.72,0.00),v40,z0,tPen\WObj:=wPaper;
    MoveL Offs(pOrigin,261.97,220.81,0.00),v40,fine,tPen\WObj:=wPaper;
    MoveL Offs(pOrigin,261.97,220.81,6.00),v60,z5,tPen\WObj:=wPaper;
    MoveL Offs(pOrigin,253.99,231.51,6.00),vTravel,z5,tPen\WObj:=wPaper;
    MoveL Offs(pOrigin,253.99,231.51,0.00),v60,z0,tPen\WObj:=wPaper;
    MoveL Offs(pOrigin,255.27,234.86,0.00),v40,z0,tPen\WObj:=wPaper;
    MoveL Offs(pOrigin,255.27,235.82,0.00),v40,z0,tPen\WObj:=wPaper;
    MoveL Offs(pOrigin,260.06,251.14,0.00),v40,z0,tPen\WObj:=wPaper;
    MoveL Offs(pOrigin,260.06,252.10,0.00),v40,z0,tPen\WObj:=wPaper;
    MoveL Offs(pOrigin,269.63,281.79,0.00),v40,z0,tPen\WObj:=wPaper;
    MoveL Offs(pOrigin,269.63,282.75,0.00),v40,z0,tPen\WObj:=wPaper;
    MoveL Offs(pOrigin,271.23,287.54,0.00),v40,z0,tPen\WObj:=wPaper;
    MoveL Offs(pOrigin,272.03,288.97,0.00),v40,z0,tPen\WObj:=wPaper;
    MoveL Offs(pOrigin,272.03,289.93,0.00),v40,z0,tPen\WObj:=wPaper;
    MoveL Offs(pOrigin,273.46,294.72,0.00),v40,z0,tPen\WObj:=wPaper;
    MoveL Offs(pOrigin,274.42,296.63,0.00),v40,z0,tPen\WObj:=wPaper;
    MoveL Offs(pOrigin,274.42,297.59,0.00),v40,z0,tPen\WObj:=wPaper;
    MoveL Offs(pOrigin,276.82,304.30,0.00),v40,z0,tPen\WObj:=wPaper;
    MoveL Offs(pOrigin,277.77,308.61,0.00),v40,z0,tPen\WObj:=wPaper;
    MoveL Offs(pOrigin,280.33,316.27,0.00),v40,z0,tPen\WObj:=wPaper;
    MoveL Offs(pOrigin,253.99,231.51,0.00),v40,fine,tPen\WObj:=wPaper;
    MoveL Offs(pOrigin,253.99,231.51,6.00),v60,z5,tPen\WObj:=wPaper;
    MoveL Offs(pOrigin,264.37,242.04,6.00),vTravel,z5,tPen\WObj:=wPaper;
    MoveL Offs(pOrigin,264.37,242.04,0.00),v60,z0,tPen\WObj:=wPaper;
    MoveL Offs(pOrigin,264.37,242.52,0.00),v40,z0,tPen\WObj:=wPaper;
    MoveL Offs(pOrigin,264.85,243.00,0.00),v40,z0,tPen\WObj:=wPaper;
    MoveL Offs(pOrigin,264.37,242.04,0.00),v40,z0,tPen\WObj:=wPaper;
    MoveL Offs(pOrigin,264.37,242.52,0.00),v40,z0,tPen\WObj:=wPaper;
    MoveL Offs(pOrigin,264.85,243.00,0.00),v40,z0,tPen\WObj:=wPaper;
    MoveL Offs(pOrigin,264.37,242.04,0.00),v40,fine,tPen\WObj:=wPaper;
    MoveL Offs(pOrigin,264.37,242.04,6.00),v60,z5,tPen\WObj:=wPaper;
    MoveL Offs(pOrigin,276.50,227.04,6.00),vTravel,z5,tPen\WObj:=wPaper;
    MoveL Offs(pOrigin,276.50,227.04,0.00),v60,z0,tPen\WObj:=wPaper;
    MoveL Offs(pOrigin,287.83,232.15,0.00),v40,z0,tPen\WObj:=wPaper;
    MoveL Offs(pOrigin,316.08,243.80,0.00),v40,z0,tPen\WObj:=wPaper;
    MoveL Offs(pOrigin,327.58,249.07,0.00),v40,z0,tPen\WObj:=wPaper;
    MoveL Offs(pOrigin,329.01,249.38,0.00),v40,z0,tPen\WObj:=wPaper;
    MoveL Offs(pOrigin,332.85,251.30,0.00),v40,z0,tPen\WObj:=wPaper;
    MoveL Offs(pOrigin,343.86,255.61,0.00),v40,z0,tPen\WObj:=wPaper;
    MoveL Offs(pOrigin,355.83,261.04,0.00),v40,z0,tPen\WObj:=wPaper;
    MoveL Offs(pOrigin,361.10,262.95,0.00),v40,z0,tPen\WObj:=wPaper;
    MoveL Offs(pOrigin,363.81,264.55,0.00),v40,z0,tPen\WObj:=wPaper;
    MoveL Offs(pOrigin,363.81,266.94,0.00),v40,z0,tPen\WObj:=wPaper;
    MoveL Offs(pOrigin,362.22,269.50,0.00),v40,z0,tPen\WObj:=wPaper;
    MoveL Offs(pOrigin,360.78,272.69,0.00),v40,z0,tPen\WObj:=wPaper;
    MoveL Offs(pOrigin,359.50,274.13,0.00),v40,z0,tPen\WObj:=wPaper;
    MoveL Offs(pOrigin,359.02,275.56,0.00),v40,z0,tPen\WObj:=wPaper;
    MoveL Offs(pOrigin,357.43,277.64,0.00),v40,z0,tPen\WObj:=wPaper;
    MoveL Offs(pOrigin,356.63,279.39,0.00),v40,z0,tPen\WObj:=wPaper;
    MoveL Offs(pOrigin,355.51,280.35,0.00),v40,z0,tPen\WObj:=wPaper;
    MoveL Offs(pOrigin,354.23,282.75,0.00),v40,z0,tPen\WObj:=wPaper;
    MoveL Offs(pOrigin,353.12,283.70,0.00),v40,z0,tPen\WObj:=wPaper;
    MoveL Offs(pOrigin,351.36,286.58,0.00),v40,z0,tPen\WObj:=wPaper;
    MoveL Offs(pOrigin,350.24,287.54,0.00),v40,z0,tPen\WObj:=wPaper;
    MoveL Offs(pOrigin,349.92,288.49,0.00),v40,z0,tPen\WObj:=wPaper;
    MoveL Offs(pOrigin,347.37,290.89,0.00),v40,z0,tPen\WObj:=wPaper;
    MoveL Offs(pOrigin,346.09,292.80,0.00),v40,z0,tPen\WObj:=wPaper;
    MoveL Offs(pOrigin,344.02,294.88,0.00),v40,z0,tPen\WObj:=wPaper;
    MoveL Offs(pOrigin,343.70,295.68,0.00),v40,z0,tPen\WObj:=wPaper;
    MoveL Offs(pOrigin,339.07,300.31,0.00),v40,z0,tPen\WObj:=wPaper;
    MoveL Offs(pOrigin,337.63,301.10,0.00),v40,z0,tPen\WObj:=wPaper;
    MoveL Offs(pOrigin,333.80,305.09,0.00),v40,z0,tPen\WObj:=wPaper;
    MoveL Offs(pOrigin,332.85,305.41,0.00),v40,z0,tPen\WObj:=wPaper;
    MoveL Offs(pOrigin,330.45,307.97,0.00),v40,z0,tPen\WObj:=wPaper;
    MoveL Offs(pOrigin,329.49,308.29,0.00),v40,z0,tPen\WObj:=wPaper;
    MoveL Offs(pOrigin,328.54,309.40,0.00),v40,z0,tPen\WObj:=wPaper;
    MoveL Offs(pOrigin,327.58,309.72,0.00),v40,z0,tPen\WObj:=wPaper;
    MoveL Offs(pOrigin,326.62,310.84,0.00),v40,z0,tPen\WObj:=wPaper;
    MoveL Offs(pOrigin,325.18,311.64,0.00),v40,z0,tPen\WObj:=wPaper;
    MoveL Offs(pOrigin,324.23,312.76,0.00),v40,z0,tPen\WObj:=wPaper;
    MoveL Offs(pOrigin,323.27,313.08,0.00),v40,z0,tPen\WObj:=wPaper;
    MoveL Offs(pOrigin,322.95,313.55,0.00),v40,z0,tPen\WObj:=wPaper;
    MoveL Offs(pOrigin,276.50,227.04,0.00),v40,fine,tPen\WObj:=wPaper;
    MoveL Offs(pOrigin,276.50,227.04,6.00),v60,z5,tPen\WObj:=wPaper;
    MoveL Offs(pOrigin,284.48,249.07,6.00),vTravel,z5,tPen\WObj:=wPaper;
    MoveL Offs(pOrigin,284.48,249.07,0.00),v60,z0,tPen\WObj:=wPaper;
    MoveL Offs(pOrigin,283.04,249.86,0.00),v40,z0,tPen\WObj:=wPaper;
    MoveL Offs(pOrigin,281.29,251.62,0.00),v40,z0,tPen\WObj:=wPaper;
    MoveL Offs(pOrigin,280.33,253.54,0.00),v40,z0,tPen\WObj:=wPaper;
    MoveL Offs(pOrigin,279.37,254.65,0.00),v40,z0,tPen\WObj:=wPaper;
    MoveL Offs(pOrigin,278.73,257.37,0.00),v40,z0,tPen\WObj:=wPaper;
    MoveL Offs(pOrigin,278.73,260.24,0.00),v40,z0,tPen\WObj:=wPaper;
    MoveL Offs(pOrigin,280.01,265.03,0.00),v40,z0,tPen\WObj:=wPaper;
    MoveL Offs(pOrigin,282.40,267.90,0.00),v40,z0,tPen\WObj:=wPaper;
    MoveL Offs(pOrigin,284.48,269.66,0.00),v40,z0,tPen\WObj:=wPaper;
    MoveL Offs(pOrigin,287.35,270.77,0.00),v40,z0,tPen\WObj:=wPaper;
    MoveL Offs(pOrigin,292.62,270.77,0.00),v40,z0,tPen\WObj:=wPaper;
    MoveL Offs(pOrigin,295.97,269.66,0.00),v40,z0,tPen\WObj:=wPaper;
    MoveL Offs(pOrigin,297.89,268.38,0.00),v40,z0,tPen\WObj:=wPaper;
    MoveL Offs(pOrigin,300.44,265.03,0.00),v40,z0,tPen\WObj:=wPaper;
    MoveL Offs(pOrigin,301.72,261.20,0.00),v40,z0,tPen\WObj:=wPaper;
    MoveL Offs(pOrigin,301.72,257.85,0.00),v40,z0,tPen\WObj:=wPaper;
    MoveL Offs(pOrigin,300.60,254.49,0.00),v40,z0,tPen\WObj:=wPaper;
    MoveL Offs(pOrigin,298.85,251.62,0.00),v40,z0,tPen\WObj:=wPaper;
    MoveL Offs(pOrigin,295.49,249.07,0.00),v40,z0,tPen\WObj:=wPaper;
    MoveL Offs(pOrigin,293.10,248.27,0.00),v40,z0,tPen\WObj:=wPaper;
    MoveL Offs(pOrigin,291.66,248.27,0.00),v40,z0,tPen\WObj:=wPaper;
    MoveL Offs(pOrigin,290.23,247.79,0.00),v40,z0,tPen\WObj:=wPaper;
    MoveL Offs(pOrigin,286.87,248.27,0.00),v40,z0,tPen\WObj:=wPaper;
  ENDPROC

  PROC DrawPart21()
    MoveL Offs(pOrigin,284.48,249.07,0.00),v40,z0,tPen\WObj:=wPaper;
    MoveL Offs(pOrigin,284.48,249.23,0.00),v40,z0,tPen\WObj:=wPaper;
    MoveL Offs(pOrigin,284.96,249.23,0.00),v40,z0,tPen\WObj:=wPaper;
    MoveL Offs(pOrigin,284.00,249.70,0.00),v40,z0,tPen\WObj:=wPaper;
    MoveL Offs(pOrigin,284.48,249.23,0.00),v40,z0,tPen\WObj:=wPaper;
    MoveL Offs(pOrigin,284.96,249.23,0.00),v40,z0,tPen\WObj:=wPaper;
    MoveL Offs(pOrigin,284.00,249.70,0.00),v40,z0,tPen\WObj:=wPaper;
    MoveL Offs(pOrigin,284.48,249.23,0.00),v40,fine,tPen\WObj:=wPaper;
    MoveL Offs(pOrigin,284.48,249.23,6.00),v60,z5,tPen\WObj:=wPaper;
    MoveL Offs(pOrigin,282.08,250.66,6.00),vTravel,z5,tPen\WObj:=wPaper;
    MoveL Offs(pOrigin,282.08,250.66,0.00),v60,z0,tPen\WObj:=wPaper;
    MoveL Offs(pOrigin,282.08,251.14,0.00),v40,z0,tPen\WObj:=wPaper;
    MoveL Offs(pOrigin,281.61,251.62,0.00),v40,z0,tPen\WObj:=wPaper;
    MoveL Offs(pOrigin,282.08,250.66,0.00),v40,z0,tPen\WObj:=wPaper;
    MoveL Offs(pOrigin,282.08,251.14,0.00),v40,z0,tPen\WObj:=wPaper;
    MoveL Offs(pOrigin,281.61,251.62,0.00),v40,z0,tPen\WObj:=wPaper;
    MoveL Offs(pOrigin,282.08,250.66,0.00),v40,fine,tPen\WObj:=wPaper;
    MoveL Offs(pOrigin,282.08,250.66,6.00),v60,z5,tPen\WObj:=wPaper;
    MoveL Offs(pOrigin,295.01,249.23,6.00),vTravel,z5,tPen\WObj:=wPaper;
    MoveL Offs(pOrigin,295.01,249.23,0.00),v60,z0,tPen\WObj:=wPaper;
    MoveL Offs(pOrigin,295.49,249.23,0.00),v40,z0,tPen\WObj:=wPaper;
    MoveL Offs(pOrigin,296.45,250.18,0.00),v40,z0,tPen\WObj:=wPaper;
    MoveL Offs(pOrigin,295.01,249.23,0.00),v40,z0,tPen\WObj:=wPaper;
    MoveL Offs(pOrigin,295.49,249.23,0.00),v40,z0,tPen\WObj:=wPaper;
    MoveL Offs(pOrigin,296.45,250.18,0.00),v40,z0,tPen\WObj:=wPaper;
    MoveL Offs(pOrigin,295.01,249.23,0.00),v40,fine,tPen\WObj:=wPaper;
    MoveL Offs(pOrigin,295.01,249.23,6.00),v60,z5,tPen\WObj:=wPaper;
    MoveL Offs(pOrigin,296.45,243.48,6.00),vTravel,z5,tPen\WObj:=wPaper;
    MoveL Offs(pOrigin,296.45,243.48,0.00),v60,z0,tPen\WObj:=wPaper;
    MoveL Offs(pOrigin,295.49,243.00,0.00),v40,z0,tPen\WObj:=wPaper;
    MoveL Offs(pOrigin,295.97,243.00,0.00),v40,z0,tPen\WObj:=wPaper;
    MoveL Offs(pOrigin,296.45,243.48,0.00),v40,z0,tPen\WObj:=wPaper;
    MoveL Offs(pOrigin,295.49,243.00,0.00),v40,z0,tPen\WObj:=wPaper;
    MoveL Offs(pOrigin,295.97,243.00,0.00),v40,z0,tPen\WObj:=wPaper;
    MoveL Offs(pOrigin,296.45,243.48,0.00),v40,fine,tPen\WObj:=wPaper;
    MoveL Offs(pOrigin,296.45,243.48,6.00),v60,z5,tPen\WObj:=wPaper;
    MoveL Offs(pOrigin,301.24,245.39,6.00),vTravel,z5,tPen\WObj:=wPaper;
    MoveL Offs(pOrigin,301.24,245.39,0.00),v60,z0,tPen\WObj:=wPaper;
    MoveL Offs(pOrigin,301.72,245.39,0.00),v40,z0,tPen\WObj:=wPaper;
    MoveL Offs(pOrigin,302.20,245.87,0.00),v40,z0,tPen\WObj:=wPaper;
    MoveL Offs(pOrigin,301.24,245.39,0.00),v40,z0,tPen\WObj:=wPaper;
    MoveL Offs(pOrigin,301.72,245.39,0.00),v40,z0,tPen\WObj:=wPaper;
    MoveL Offs(pOrigin,302.20,245.87,0.00),v40,z0,tPen\WObj:=wPaper;
    MoveL Offs(pOrigin,301.24,245.39,0.00),v40,fine,tPen\WObj:=wPaper;
    MoveL Offs(pOrigin,301.24,245.39,6.00),v60,z5,tPen\WObj:=wPaper;
    MoveL Offs(pOrigin,307.46,248.27,6.00),vTravel,z5,tPen\WObj:=wPaper;
    MoveL Offs(pOrigin,307.46,248.27,0.00),v60,z0,tPen\WObj:=wPaper;
    MoveL Offs(pOrigin,307.94,248.27,0.00),v40,z0,tPen\WObj:=wPaper;
    MoveL Offs(pOrigin,308.42,248.75,0.00),v40,z0,tPen\WObj:=wPaper;
    MoveL Offs(pOrigin,307.46,248.27,0.00),v40,z0,tPen\WObj:=wPaper;
    MoveL Offs(pOrigin,307.94,248.27,0.00),v40,z0,tPen\WObj:=wPaper;
    MoveL Offs(pOrigin,308.42,248.75,0.00),v40,z0,tPen\WObj:=wPaper;
    MoveL Offs(pOrigin,307.46,248.27,0.00),v40,fine,tPen\WObj:=wPaper;
    MoveL Offs(pOrigin,307.46,248.27,6.00),v60,z5,tPen\WObj:=wPaper;
    MoveL Offs(pOrigin,321.83,254.97,6.00),vTravel,z5,tPen\WObj:=wPaper;
    MoveL Offs(pOrigin,321.83,254.97,0.00),v60,z0,tPen\WObj:=wPaper;
    MoveL Offs(pOrigin,322.31,254.97,0.00),v40,z0,tPen\WObj:=wPaper;
    MoveL Offs(pOrigin,322.79,255.45,0.00),v40,z0,tPen\WObj:=wPaper;
    MoveL Offs(pOrigin,321.83,254.97,0.00),v40,z0,tPen\WObj:=wPaper;
    MoveL Offs(pOrigin,322.31,254.97,0.00),v40,z0,tPen\WObj:=wPaper;
    MoveL Offs(pOrigin,322.79,255.45,0.00),v40,z0,tPen\WObj:=wPaper;
    MoveL Offs(pOrigin,321.83,254.97,0.00),v40,fine,tPen\WObj:=wPaper;
    MoveL Offs(pOrigin,321.83,254.97,6.00),v60,z5,tPen\WObj:=wPaper;
    MoveL Offs(pOrigin,321.83,261.68,6.00),vTravel,z5,tPen\WObj:=wPaper;
    MoveL Offs(pOrigin,321.83,261.68,0.00),v60,z0,tPen\WObj:=wPaper;
    MoveL Offs(pOrigin,323.27,261.68,0.00),v40,z0,tPen\WObj:=wPaper;
    MoveL Offs(pOrigin,327.10,262.79,0.00),v40,z0,tPen\WObj:=wPaper;
    MoveL Offs(pOrigin,329.81,264.71,0.00),v40,z0,tPen\WObj:=wPaper;
    MoveL Offs(pOrigin,329.49,264.07,0.00),v40,z0,tPen\WObj:=wPaper;
    MoveL Offs(pOrigin,318.00,262.95,0.00),v40,z0,tPen\WObj:=wPaper;
    MoveL Offs(pOrigin,321.83,261.68,0.00),v40,fine,tPen\WObj:=wPaper;
    MoveL Offs(pOrigin,321.83,261.68,6.00),v60,z5,tPen\WObj:=wPaper;
    MoveL Offs(pOrigin,317.04,263.11,6.00),vTravel,z5,tPen\WObj:=wPaper;
    MoveL Offs(pOrigin,317.04,263.11,0.00),v60,z0,tPen\WObj:=wPaper;
    MoveL Offs(pOrigin,316.08,264.07,0.00),v40,z0,tPen\WObj:=wPaper;
    MoveL Offs(pOrigin,316.56,264.07,0.00),v40,z0,tPen\WObj:=wPaper;
    MoveL Offs(pOrigin,317.04,263.59,0.00),v40,z0,tPen\WObj:=wPaper;
    MoveL Offs(pOrigin,317.04,263.11,0.00),v40,z0,tPen\WObj:=wPaper;
    MoveL Offs(pOrigin,316.08,264.07,0.00),v40,z0,tPen\WObj:=wPaper;
    MoveL Offs(pOrigin,316.56,264.07,0.00),v40,z0,tPen\WObj:=wPaper;
    MoveL Offs(pOrigin,317.04,263.59,0.00),v40,z0,tPen\WObj:=wPaper;
    MoveL Offs(pOrigin,317.04,263.11,0.00),v40,fine,tPen\WObj:=wPaper;
    MoveL Offs(pOrigin,317.04,263.11,6.00),v60,z5,tPen\WObj:=wPaper;
    MoveL Offs(pOrigin,315.45,264.55,6.00),vTravel,z5,tPen\WObj:=wPaper;
    MoveL Offs(pOrigin,315.45,264.55,0.00),v60,z0,tPen\WObj:=wPaper;
    MoveL Offs(pOrigin,312.89,266.94,0.00),v40,z0,tPen\WObj:=wPaper;
    MoveL Offs(pOrigin,312.57,268.38,0.00),v40,z0,tPen\WObj:=wPaper;
    MoveL Offs(pOrigin,311.77,269.34,0.00),v40,z0,tPen\WObj:=wPaper;
    MoveL Offs(pOrigin,311.30,271.73,0.00),v40,z0,tPen\WObj:=wPaper;
    MoveL Offs(pOrigin,311.30,274.61,0.00),v40,z0,tPen\WObj:=wPaper;
    MoveL Offs(pOrigin,311.77,277.00,0.00),v40,z0,tPen\WObj:=wPaper;
    MoveL Offs(pOrigin,312.57,278.92,0.00),v40,z0,tPen\WObj:=wPaper;
    MoveL Offs(pOrigin,314.49,281.47,0.00),v40,z0,tPen\WObj:=wPaper;
    MoveL Offs(pOrigin,315.45,264.55,0.00),v40,z0,tPen\WObj:=wPaper;
    MoveL Offs(pOrigin,315.13,264.55,0.00),v40,z0,tPen\WObj:=wPaper;
    MoveL Offs(pOrigin,314.65,265.51,0.00),v40,z0,tPen\WObj:=wPaper;
    MoveL Offs(pOrigin,315.13,265.03,0.00),v40,z0,tPen\WObj:=wPaper;
    MoveL Offs(pOrigin,315.13,264.55,0.00),v40,z0,tPen\WObj:=wPaper;
    MoveL Offs(pOrigin,314.65,265.51,0.00),v40,z0,tPen\WObj:=wPaper;
    MoveL Offs(pOrigin,315.13,265.03,0.00),v40,z0,tPen\WObj:=wPaper;
    MoveL Offs(pOrigin,315.13,264.55,0.00),v40,fine,tPen\WObj:=wPaper;
    MoveL Offs(pOrigin,315.13,264.55,6.00),v60,z5,tPen\WObj:=wPaper;
    MoveL Offs(pOrigin,313.69,265.99,6.00),vTravel,z5,tPen\WObj:=wPaper;
    MoveL Offs(pOrigin,313.69,265.99,0.00),v60,z0,tPen\WObj:=wPaper;
    MoveL Offs(pOrigin,313.21,266.94,0.00),v40,z0,tPen\WObj:=wPaper;
    MoveL Offs(pOrigin,313.69,266.46,0.00),v40,z0,tPen\WObj:=wPaper;
    MoveL Offs(pOrigin,313.69,265.99,0.00),v40,z0,tPen\WObj:=wPaper;
    MoveL Offs(pOrigin,313.21,266.94,0.00),v40,z0,tPen\WObj:=wPaper;
    MoveL Offs(pOrigin,313.69,266.46,0.00),v40,z0,tPen\WObj:=wPaper;
    MoveL Offs(pOrigin,313.69,265.99,0.00),v40,fine,tPen\WObj:=wPaper;
    MoveL Offs(pOrigin,313.69,265.99,6.00),v60,z5,tPen\WObj:=wPaper;
    MoveL Offs(pOrigin,312.25,277.48,6.00),vTravel,z5,tPen\WObj:=wPaper;
    MoveL Offs(pOrigin,312.25,277.48,0.00),v60,z0,tPen\WObj:=wPaper;
    MoveL Offs(pOrigin,312.25,277.96,0.00),v40,z0,tPen\WObj:=wPaper;
    MoveL Offs(pOrigin,312.73,278.44,0.00),v40,z0,tPen\WObj:=wPaper;
    MoveL Offs(pOrigin,312.25,277.48,0.00),v40,z0,tPen\WObj:=wPaper;
    MoveL Offs(pOrigin,312.25,277.96,0.00),v40,z0,tPen\WObj:=wPaper;
    MoveL Offs(pOrigin,312.73,278.44,0.00),v40,z0,tPen\WObj:=wPaper;
    MoveL Offs(pOrigin,312.25,277.48,0.00),v40,fine,tPen\WObj:=wPaper;
    MoveL Offs(pOrigin,312.25,277.48,6.00),v60,z5,tPen\WObj:=wPaper;
  ENDPROC

  PROC DrawPart22()
    MoveL Offs(pOrigin,313.21,279.39,6.00),vTravel,z5,tPen\WObj:=wPaper;
    MoveL Offs(pOrigin,313.21,279.39,0.00),v60,z0,tPen\WObj:=wPaper;
    MoveL Offs(pOrigin,313.21,279.87,0.00),v40,z0,tPen\WObj:=wPaper;
    MoveL Offs(pOrigin,313.69,279.87,0.00),v40,z0,tPen\WObj:=wPaper;
    MoveL Offs(pOrigin,313.21,279.39,0.00),v40,z0,tPen\WObj:=wPaper;
    MoveL Offs(pOrigin,313.21,279.87,0.00),v40,z0,tPen\WObj:=wPaper;
    MoveL Offs(pOrigin,313.69,279.87,0.00),v40,z0,tPen\WObj:=wPaper;
    MoveL Offs(pOrigin,313.21,279.39,0.00),v40,fine,tPen\WObj:=wPaper;
    MoveL Offs(pOrigin,313.21,279.39,6.00),v60,z5,tPen\WObj:=wPaper;
    MoveL Offs(pOrigin,315.29,282.27,6.00),vTravel,z5,tPen\WObj:=wPaper;
    MoveL Offs(pOrigin,315.29,282.27,0.00),v60,z0,tPen\WObj:=wPaper;
    MoveL Offs(pOrigin,317.52,284.02,0.00),v40,z0,tPen\WObj:=wPaper;
    MoveL Offs(pOrigin,320.39,285.14,0.00),v40,z0,tPen\WObj:=wPaper;
    MoveL Offs(pOrigin,325.18,285.14,0.00),v40,z0,tPen\WObj:=wPaper;
    MoveL Offs(pOrigin,327.10,284.34,0.00),v40,z0,tPen\WObj:=wPaper;
    MoveL Offs(pOrigin,323.27,283.38,0.00),v40,z0,tPen\WObj:=wPaper;
    MoveL Offs(pOrigin,315.29,282.27,0.00),v40,fine,tPen\WObj:=wPaper;
    MoveL Offs(pOrigin,315.29,282.27,6.00),v60,z5,tPen\WObj:=wPaper;
    MoveL Offs(pOrigin,310.82,285.14,6.00),vTravel,z5,tPen\WObj:=wPaper;
    MoveL Offs(pOrigin,310.82,285.14,0.00),v60,z0,tPen\WObj:=wPaper;
    MoveL Offs(pOrigin,309.38,283.23,0.00),v40,z0,tPen\WObj:=wPaper;
    MoveL Offs(pOrigin,309.38,283.70,0.00),v40,z0,tPen\WObj:=wPaper;
    MoveL Offs(pOrigin,310.82,285.14,0.00),v40,z0,tPen\WObj:=wPaper;
    MoveL Offs(pOrigin,309.38,283.23,0.00),v40,z0,tPen\WObj:=wPaper;
    MoveL Offs(pOrigin,309.38,283.70,0.00),v40,z0,tPen\WObj:=wPaper;
    MoveL Offs(pOrigin,310.82,285.14,0.00),v40,z0,tPen\WObj:=wPaper;
    MoveL Offs(pOrigin,310.82,285.62,0.00),v40,z0,tPen\WObj:=wPaper;
    MoveL Offs(pOrigin,293.74,281.47,0.00),v40,z0,tPen\WObj:=wPaper;
    MoveL Offs(pOrigin,297.89,279.39,0.00),v40,z0,tPen\WObj:=wPaper;
    MoveL Offs(pOrigin,302.68,279.39,0.00),v40,z0,tPen\WObj:=wPaper;
    MoveL Offs(pOrigin,305.55,280.51,0.00),v40,z0,tPen\WObj:=wPaper;
    MoveL Offs(pOrigin,307.94,282.27,0.00),v40,z0,tPen\WObj:=wPaper;
    MoveL Offs(pOrigin,310.82,285.62,0.00),v40,z0,tPen\WObj:=wPaper;
    MoveL Offs(pOrigin,311.30,286.58,0.00),v40,z0,tPen\WObj:=wPaper;
    MoveL Offs(pOrigin,312.73,291.37,0.00),v40,z0,tPen\WObj:=wPaper;
    MoveL Offs(pOrigin,311.77,295.68,0.00),v40,z0,tPen\WObj:=wPaper;
    MoveL Offs(pOrigin,310.18,298.55,0.00),v40,z0,tPen\WObj:=wPaper;
    MoveL Offs(pOrigin,307.62,301.10,0.00),v40,z0,tPen\WObj:=wPaper;
    MoveL Offs(pOrigin,311.30,286.58,0.00),v40,fine,tPen\WObj:=wPaper;
    MoveL Offs(pOrigin,311.30,286.58,6.00),v60,z5,tPen\WObj:=wPaper;
    MoveL Offs(pOrigin,308.90,282.75,6.00),vTravel,z5,tPen\WObj:=wPaper;
    MoveL Offs(pOrigin,308.90,282.75,0.00),v60,z0,tPen\WObj:=wPaper;
    MoveL Offs(pOrigin,307.94,281.79,0.00),v40,z0,tPen\WObj:=wPaper;
    MoveL Offs(pOrigin,307.94,282.27,0.00),v40,z0,tPen\WObj:=wPaper;
    MoveL Offs(pOrigin,308.42,282.27,0.00),v40,z0,tPen\WObj:=wPaper;
    MoveL Offs(pOrigin,308.90,282.75,0.00),v40,z0,tPen\WObj:=wPaper;
    MoveL Offs(pOrigin,307.94,281.79,0.00),v40,z0,tPen\WObj:=wPaper;
    MoveL Offs(pOrigin,307.94,282.27,0.00),v40,z0,tPen\WObj:=wPaper;
    MoveL Offs(pOrigin,308.42,282.27,0.00),v40,z0,tPen\WObj:=wPaper;
    MoveL Offs(pOrigin,308.90,282.75,0.00),v40,fine,tPen\WObj:=wPaper;
    MoveL Offs(pOrigin,308.90,282.75,6.00),v60,z5,tPen\WObj:=wPaper;
    MoveL Offs(pOrigin,306.99,281.31,6.00),vTravel,z5,tPen\WObj:=wPaper;
    MoveL Offs(pOrigin,306.99,281.31,0.00),v60,z0,tPen\WObj:=wPaper;
    MoveL Offs(pOrigin,306.51,280.83,0.00),v40,z0,tPen\WObj:=wPaper;
    MoveL Offs(pOrigin,306.51,281.31,0.00),v40,z0,tPen\WObj:=wPaper;
    MoveL Offs(pOrigin,306.99,281.31,0.00),v40,z0,tPen\WObj:=wPaper;
    MoveL Offs(pOrigin,306.51,280.83,0.00),v40,z0,tPen\WObj:=wPaper;
    MoveL Offs(pOrigin,306.51,281.31,0.00),v40,z0,tPen\WObj:=wPaper;
    MoveL Offs(pOrigin,306.99,281.31,0.00),v40,fine,tPen\WObj:=wPaper;
    MoveL Offs(pOrigin,306.99,281.31,6.00),v60,z5,tPen\WObj:=wPaper;
    MoveL Offs(pOrigin,293.10,281.79,6.00),vTravel,z5,tPen\WObj:=wPaper;
    MoveL Offs(pOrigin,293.10,281.79,0.00),v60,z0,tPen\WObj:=wPaper;
    MoveL Offs(pOrigin,292.62,281.79,0.00),v40,z0,tPen\WObj:=wPaper;
    MoveL Offs(pOrigin,292.14,282.27,0.00),v40,z0,tPen\WObj:=wPaper;
    MoveL Offs(pOrigin,292.14,282.75,0.00),v40,z0,tPen\WObj:=wPaper;
    MoveL Offs(pOrigin,293.10,281.79,0.00),v40,z0,tPen\WObj:=wPaper;
    MoveL Offs(pOrigin,292.62,281.79,0.00),v40,z0,tPen\WObj:=wPaper;
    MoveL Offs(pOrigin,292.14,282.27,0.00),v40,z0,tPen\WObj:=wPaper;
    MoveL Offs(pOrigin,292.14,282.75,0.00),v40,z0,tPen\WObj:=wPaper;
    MoveL Offs(pOrigin,293.10,281.79,0.00),v40,fine,tPen\WObj:=wPaper;
    MoveL Offs(pOrigin,293.10,281.79,6.00),v60,z5,tPen\WObj:=wPaper;
    MoveL Offs(pOrigin,291.50,283.23,6.00),vTravel,z5,tPen\WObj:=wPaper;
    MoveL Offs(pOrigin,291.50,283.23,0.00),v60,z0,tPen\WObj:=wPaper;
    MoveL Offs(pOrigin,289.91,285.62,0.00),v40,z0,tPen\WObj:=wPaper;
    MoveL Offs(pOrigin,289.59,287.06,0.00),v40,z0,tPen\WObj:=wPaper;
    MoveL Offs(pOrigin,288.95,288.01,0.00),v40,z0,tPen\WObj:=wPaper;
    MoveL Offs(pOrigin,291.50,283.23,0.00),v40,fine,tPen\WObj:=wPaper;
    MoveL Offs(pOrigin,291.50,283.23,6.00),v60,z5,tPen\WObj:=wPaper;
    MoveL Offs(pOrigin,288.79,288.97,6.00),vTravel,z5,tPen\WObj:=wPaper;
    MoveL Offs(pOrigin,288.79,288.97,0.00),v60,z0,tPen\WObj:=wPaper;
    MoveL Offs(pOrigin,288.79,290.41,0.00),v40,z0,tPen\WObj:=wPaper;
    MoveL Offs(pOrigin,288.79,288.97,0.00),v40,fine,tPen\WObj:=wPaper;
    MoveL Offs(pOrigin,288.79,288.97,6.00),v60,z5,tPen\WObj:=wPaper;
    MoveL Offs(pOrigin,288.79,291.37,6.00),vTravel,z5,tPen\WObj:=wPaper;
    MoveL Offs(pOrigin,288.79,291.37,0.00),v60,z0,tPen\WObj:=wPaper;
    MoveL Offs(pOrigin,288.79,293.76,0.00),v40,z0,tPen\WObj:=wPaper;
    MoveL Offs(pOrigin,290.07,297.11,0.00),v40,z0,tPen\WObj:=wPaper;
    MoveL Offs(pOrigin,291.66,299.51,0.00),v40,z0,tPen\WObj:=wPaper;
    MoveL Offs(pOrigin,294.54,301.74,0.00),v40,z0,tPen\WObj:=wPaper;
    MoveL Offs(pOrigin,296.45,302.70,0.00),v40,z0,tPen\WObj:=wPaper;
    MoveL Offs(pOrigin,298.85,303.34,0.00),v40,z0,tPen\WObj:=wPaper;
    MoveL Offs(pOrigin,302.68,303.34,0.00),v40,z0,tPen\WObj:=wPaper;
    MoveL Offs(pOrigin,305.07,302.54,0.00),v40,z0,tPen\WObj:=wPaper;
    MoveL Offs(pOrigin,306.67,301.58,0.00),v40,z0,tPen\WObj:=wPaper;
    MoveL Offs(pOrigin,300.76,297.91,0.00),v40,z0,tPen\WObj:=wPaper;
    MoveL Offs(pOrigin,288.79,291.37,0.00),v40,fine,tPen\WObj:=wPaper;
    MoveL Offs(pOrigin,288.79,291.37,6.00),v60,z5,tPen\WObj:=wPaper;
    MoveL Offs(pOrigin,290.70,297.59,6.00),vTravel,z5,tPen\WObj:=wPaper;
    MoveL Offs(pOrigin,290.70,297.59,0.00),v60,z0,tPen\WObj:=wPaper;
    MoveL Offs(pOrigin,290.70,298.07,0.00),v40,z0,tPen\WObj:=wPaper;
    MoveL Offs(pOrigin,291.18,298.07,0.00),v40,z0,tPen\WObj:=wPaper;
    MoveL Offs(pOrigin,290.70,297.59,0.00),v40,z0,tPen\WObj:=wPaper;
    MoveL Offs(pOrigin,290.70,298.07,0.00),v40,z0,tPen\WObj:=wPaper;
    MoveL Offs(pOrigin,291.18,298.07,0.00),v40,z0,tPen\WObj:=wPaper;
    MoveL Offs(pOrigin,290.70,297.59,0.00),v40,fine,tPen\WObj:=wPaper;
    MoveL Offs(pOrigin,290.70,297.59,6.00),v60,z5,tPen\WObj:=wPaper;
    MoveL Offs(pOrigin,291.66,299.03,6.00),vTravel,z5,tPen\WObj:=wPaper;
    MoveL Offs(pOrigin,291.66,299.03,0.00),v60,z0,tPen\WObj:=wPaper;
    MoveL Offs(pOrigin,291.66,299.51,0.00),v40,z0,tPen\WObj:=wPaper;
    MoveL Offs(pOrigin,292.14,299.51,0.00),v40,z0,tPen\WObj:=wPaper;
    MoveL Offs(pOrigin,293.10,300.46,0.00),v40,z0,tPen\WObj:=wPaper;
    MoveL Offs(pOrigin,291.66,299.03,0.00),v40,z0,tPen\WObj:=wPaper;
    MoveL Offs(pOrigin,291.66,299.51,0.00),v40,z0,tPen\WObj:=wPaper;
    MoveL Offs(pOrigin,292.14,299.51,0.00),v40,z0,tPen\WObj:=wPaper;
    MoveL Offs(pOrigin,293.10,300.46,0.00),v40,z0,tPen\WObj:=wPaper;
    MoveL Offs(pOrigin,291.66,299.03,0.00),v40,fine,tPen\WObj:=wPaper;
    MoveL Offs(pOrigin,291.66,299.03,6.00),v60,z5,tPen\WObj:=wPaper;
    MoveL Offs(pOrigin,281.61,291.85,6.00),vTravel,z5,tPen\WObj:=wPaper;
    MoveL Offs(pOrigin,281.61,291.85,0.00),v60,z0,tPen\WObj:=wPaper;
    MoveL Offs(pOrigin,281.13,290.89,0.00),v40,z0,tPen\WObj:=wPaper;
  ENDPROC

